(* CODESYS project XC300_NTPClient.project

Project tree, tasks and I/O mapping:
  XC303 : XC303, Eaton Automation, version 3.5.16.50
      unmapped channels: Output, Input
    application Application
      libraries: SysSocket23, * (System); SysCallback23, * (System); SysRtc23, * (System); Standard, 3.5.15.0 (System)
      task MainTask (cyclic, interval t#10ms, priority 1) calls PLC_PRG
      Global Variables/
        global variables Globale_Variablen
        global variables NetTime_Global
        global variables Variablen_Konfiguration
      POUs/
        Internal/
          function NetTime_Callback [ST]
          function NetTime_Concat_DT [ST]
          function NetTime_DayOfWeek [ST]
          function NetTime_SockClose [ST]
          function NetTime_SockCreate [ST]
          function block NetTime_Split_DT [IL]
        function block NetTime_RFC868_Client [ST]
        function block NetTime_RFC868_Server [ST]
        program PLC_PRG [ST]
  XV100 : XV100, Eaton Automation, version 3.5.16.60
    application Application
      libraries: SysSocket23, * (System); SysCallback23, * (System); SysRtc23, * (System); Standard, 3.5.15.0 (System)
      task MainTask (cyclic, interval t#10ms, priority 1) calls PLC_PRG
      Global Variables/
        global variables Globale_Variablen
        global variables NetTime_Global
        global variables Variablen_Konfiguration
      POUs/
        Internal/
          function NetTime_Callback [ST]
          function NetTime_Concat_DT [ST]
          function NetTime_DayOfWeek [ST]
          function NetTime_SockClose [ST]
          function NetTime_SockCreate [ST]
          function block NetTime_Split_DT [IL]
        function block NetTime_RFC868_Client [ST]
        function block NetTime_RFC868_Server [ST]
        program PLC_PRG [ST]
  XV300 : XV300, Eaton Automation, version 3.5.16.60
    application Application
      libraries: SysSocket23, * (System); SysCallback23, * (System); SysRtc23, * (System); Standard, 3.5.15.0 (System)
      task MainTask (cyclic, interval t#10ms, priority 1) calls PLC_PRG
      Global Variables/
        global variables Globale_Variablen
        global variables NetTime_Global
        global variables Variablen_Konfiguration
      POUs/
        Internal/
          function NetTime_Callback [ST]
          function NetTime_Concat_DT [ST]
          function NetTime_DayOfWeek [ST]
          function NetTime_SockClose [ST]
          function NetTime_SockCreate [ST]
          function block NetTime_Split_DT [IL]
        function block NetTime_RFC868_Client [ST]
        function block NetTime_RFC868_Server [ST]
        program PLC_PRG [ST]
*)

// XC303/Application/Global Variables/Globale_Variablen
VAR_GLOBAL
END_VAR

// XC303/Application/Global Variables/NetTime_Global
VAR_GLOBAL CONSTANT
	NetTime_striVersion 			: STRING := 'NTP V 1.0';							(* string with actual library version *)
	NetTime_iVersion_1_0		: INT;												(* variable to check compatibility *)
	NetTime_uiMaxSocketIndex 	: UINT := 10 ;										(* maximum count of sockets used in library *)
END_VAR
VAR_GLOBAL RETAIN
	NetTime_CallbackCounter : UINT ;
	NetTime_CallbackEVENT_STOPCounter : UINT ;
	NetTime_LastEvent : DWORD ;
	NetTime_LastFilter : DWORD ;
	NetTime_LastOwner : DWORD ;
END_VAR
VAR_GLOBAL
	NetTime_xCallbackRegistered : BOOL ;											(* callback function is registered *)
	NetTime_ar_udiSockets : ARRAY[1..NetTime_uiMaxSocketIndex] OF DINT ;	(* array with used socket IDs, 0 = empty *)
END_VAR

(*
Version		changes
1.0 			first version
*)

// XC303/Application/Global Variables/Variablen_Konfiguration
VAR_CONFIG
END_VAR

// XV100/Application/Global Variables/Globale_Variablen
VAR_GLOBAL
END_VAR

// XV100/Application/Global Variables/NetTime_Global
VAR_GLOBAL CONSTANT
	NetTime_striVersion 			: STRING := 'NTP V 1.0';							(* string with actual library version *)
	NetTime_iVersion_1_0		: INT;												(* variable to check compatibility *)
	NetTime_uiMaxSocketIndex 	: UINT := 10 ;										(* maximum count of sockets used in library *)
END_VAR
VAR_GLOBAL RETAIN
	NetTime_CallbackCounter : UINT ;
	NetTime_CallbackEVENT_STOPCounter : UINT ;
	NetTime_LastEvent : DWORD ;
	NetTime_LastFilter : DWORD ;
	NetTime_LastOwner : DWORD ;
END_VAR
VAR_GLOBAL
	NetTime_xCallbackRegistered : BOOL ;											(* callback function is registered *)
	NetTime_ar_udiSockets : ARRAY[1..NetTime_uiMaxSocketIndex] OF DINT ;	(* array with used socket IDs, 0 = empty *)
END_VAR

(*
Version		changes
1.0 			first version
*)

// XV100/Application/Global Variables/Variablen_Konfiguration
VAR_CONFIG
END_VAR

// XV300/Application/Global Variables/Globale_Variablen
VAR_GLOBAL
END_VAR

// XV300/Application/Global Variables/NetTime_Global
VAR_GLOBAL CONSTANT
	NetTime_striVersion 			: STRING := 'NTP V 1.0';							(* string with actual library version *)
	NetTime_iVersion_1_0		: INT;												(* variable to check compatibility *)
	NetTime_uiMaxSocketIndex 	: UINT := 10 ;										(* maximum count of sockets used in library *)
END_VAR
VAR_GLOBAL RETAIN
	NetTime_CallbackCounter : UINT ;
	NetTime_CallbackEVENT_STOPCounter : UINT ;
	NetTime_LastEvent : DWORD ;
	NetTime_LastFilter : DWORD ;
	NetTime_LastOwner : DWORD ;
END_VAR
VAR_GLOBAL
	NetTime_xCallbackRegistered : BOOL ;											(* callback function is registered *)
	NetTime_ar_udiSockets : ARRAY[1..NetTime_uiMaxSocketIndex] OF DINT ;	(* array with used socket IDs, 0 = empty *)
END_VAR

(*
Version		changes
1.0 			first version
*)

// XV300/Application/Global Variables/Variablen_Konfiguration
VAR_CONFIG
END_VAR

// XC303/Application/POUs/PLC_PRG
PROGRAM PLC_PRG
VAR
	FB_NetTime_RFC868_Client : NetTime_RFC868_Client ;
	FB_NetTime_RFC868_Server : NetTime_RFC868_Server ;
	FirstCall : BOOL := TRUE ;
END_VAR

(* Test of FB could be done with visualisation of XSoft *)

IF FirstCall THEN
	FB_NetTime_RFC868_Client.striIPAddress := '192.168.119.133' ;
	FB_NetTime_RFC868_Server.xEnable := 0 ;
END_IF
FirstCall := FALSE ;

FB_NetTime_RFC868_Client.xAskForTime;
FB_NetTime_RFC868_Client() ;

FB_NetTime_RFC868_Server() ;

END_PROGRAM

// XV100/Application/POUs/PLC_PRG
PROGRAM PLC_PRG
VAR
	FB_NetTime_RFC868_Client : NetTime_RFC868_Client ;
	FB_NetTime_RFC868_Server : NetTime_RFC868_Server ;
	FirstCall : BOOL := TRUE ;
END_VAR

(* Test of FB could be done with visualisation of XSoft *)

IF FirstCall THEN
	FB_NetTime_RFC868_Client.striIPAddress := '192.168.119.133' ;
	FB_NetTime_RFC868_Server.xEnable := TRUE ;
END_IF
FirstCall := FALSE ;

FB_NetTime_RFC868_Client.xAskForTime;
FB_NetTime_RFC868_Client() ;

FB_NetTime_RFC868_Server() ;

END_PROGRAM

// XV300/Application/POUs/PLC_PRG
PROGRAM PLC_PRG
VAR
	FB_NetTime_RFC868_Client : NetTime_RFC868_Client ;
	FB_NetTime_RFC868_Server : NetTime_RFC868_Server ;
	FirstCall : BOOL := TRUE ;
END_VAR

(* Test of FB could be done with visualisation of XSoft *)

IF FirstCall THEN
	FB_NetTime_RFC868_Client.striIPAddress := '192.168.119.248' ;
	FB_NetTime_RFC868_Server.xEnable := TRUE ;
END_IF
FirstCall := FALSE ;

FB_NetTime_RFC868_Client.xAskForTime;
FB_NetTime_RFC868_Client() ;

FB_NetTime_RFC868_Server() ;

END_PROGRAM

// XC303/Application/POUs/NetTime_RFC868_Client
FUNCTION_BLOCK NetTime_RFC868_Client
(* this FB is a client for time request to a server using a protocol described in RFC868 / UDP *)

VAR_INPUT
	striIPAddress : STRING(15) ; 				(* IP-address of th time server i.e '192.168.0.1' *)
	uiLocalPort : UINT := 1025 ;				(* local ethernet port 1-65535 see RFC1700 for assigned ports *)
	xAskForTime : BOOL ;						(* rising edge send a time request to the server *)
	siGMTOffset : SINT := 1 ;					(* time offset in h for local time-zone (-12..+12) i.e. +1 for Berlin *)
	xSummerWinterTime : BOOL := TRUE ;	(* consider Summertime from last sunday of march at 02:00 a.m.GMT to last sunday of october at 02:00 a.m.GMT *)
	xSetRTC : BOOL ;							(* set the local Real-Time-Clock to the received time from server *)
END_VAR

VAR_OUTPUT
	dtReceivedDateTime : DT := DATE_AND_TIME#2000-01-01-00:00:00 ;		(* received Date and Time from server *)
	uiReceivedSecond : UINT ;				(* received second from server (0..59) *)
	uiReceivedMinute : UINT ;				(* received minute from server (0..59) *)
	uiReceivedHour : UINT ;					(* received hour from server (0..23) *)
	uiReceivedDay : UINT :=1 ;				(* received Day from server (1..31) *)
	uiReceivedMonth : UINT :=1 ;				(* received Month from server (1..12) *)
	uiReceivedYear : UINT :=2000 ;			(* received year from server (2000..2092) *)
	uiReceivedDayOfWeek : UINT := 6 ;		(* received weekday. (1=Monday .. 7=Sunday) *)
	xSummerTime : BOOL ;					(* received Time is Summertime *)
	xActive : BOOL ;							(* waiting for an answer of the time server *)
	xError : BOOL ;							(* last request generate an error - look "uiErrornumber" for reason *)
	uiErrorNumber : UINT ;					(* reason for the last error
		0 = No error
		1 = Ethernet socket could not opend 
		2 = Ethernet socket could not binded
		3 = Transmit time request error
		4 = Ethernet receive error
		5 = Timeout - no answer from timeserver in the space of 5s *)
END_VAR

VAR
	xAskForTimeOld : BOOL ;
	iSocketIndex : UINT ;
	xBindSocket : BOOL ;
	diTraNr : DINT ;
	udiTime : UDINT ;
	struSOCKADDRESS_Receive : SOCKADDRESS ;
	diRecNr : DINT ;
	diIO : DINT ;
	dwParameterIO : DWORD ;
	arReceiveData : ARRAY[0..3] OF BYTE ;
	xRecIP : BOOL ;
	struInADDR_TimeServer : INADDR;
	striTimeServerIPAddress : STRING;

	TON_Timeout : TON := (PT:=T#5s) ;

	uiRemotePort : UINT := 37 ;
	struSOCKADDRESS_Bind : SOCKADDRESS ;
	struSOCKADDRESS_Transmit : SOCKADDRESS ;
	dwReceiveData : DWORD ;
	udiGMTSecondsSince1970 : UDINT ;
	i : USINT ;

	Split_DT : NetTime_Split_DT ;

	uiDayStartSummertime : UINT ;
	uiDayEndSummertime : UINT ;

	dtStartSummertime : DT ;
	dtEndSummertime : DT ;

	struSOCKADDRESS_Connect : SOCKADDRESS ;
	xSysSockConnect : BOOL ;
END_VAR

IF xActive THEN
	IF NetTime_ar_udiSockets[iSocketIndex] > 0 THEN
		(* waiting for an answer of the time-server *)
		(* is any data received *)
		diIO := SysSockIoctl(NetTime_ar_udiSockets[iSocketIndex], SOCKET_FIONREAD, ADR(dwParameterIO)); (* get num chars available to read *)
		IF dwParameterIO <> 0 THEN
			diRecNr := SysSockRecvFrom(NetTime_ar_udiSockets[iSocketIndex], ADR(arReceiveData), SIZEOF(arReceiveData), 0,
											 ADR(struSOCKADDRESS_Receive), SIZEOF(struSOCKADDRESS_Receive));
			IF diRecNr = -1 THEN
				uiErrorNumber := 4 ;
			ELSE
				(* check receive IP Address *)
				struInADDR_TimeServer.s_addr := struSOCKADDRESS_Receive.sin_addr ;
				xRecIP:=SysSockInetNtoa(struInADDR_TimeServer, striTimeServerIPAddress, SIZEOF(striTimeServerIPAddress)) ;
				IF struSOCKADDRESS_Receive.sin_addr = struSOCKADDRESS_Transmit.sin_addr THEN
					(* answer is coming from requested timeserver *)
					(* interpret received data *)
					(* change byte orientation *)
					dwReceiveData := 0 ;
					FOR i := 0 TO 3 DO
						dwReceiveData := SHL(dwReceiveData,8) ;
						dwReceiveData := dwReceiveData OR BYTE_TO_DWORD(arReceiveData[i]) ;
					END_FOR
					(* dwReceiveData = seconds after 1.1.1900 00:00:00 *)
					IF DWORD_TO_UDINT(dwReceiveData) >= UDINT#2208988800 THEN
						udiGMTSecondsSince1970 := DWORD_TO_UDINT(dwReceiveData) - UDINT#2208988800 ;
					ELSE
						udiGMTSecondsSince1970 := DWORD_TO_UDINT(dwReceiveData) + UDINT#2208988800 ;
					END_IF
					dtReceivedDateTime := UDINT_TO_DT(udiGMTSecondsSince1970+(UINT#3600*SINT_TO_DINT(siGMTOffset))) ;
	
					Split_DT(
						InputDT:=dtReceivedDateTime ,
						uiSecond=>uiReceivedSecond ,
						uiMinute=>uiReceivedMinute ,
						uiHour=>uiReceivedHour ,
						uiDay=>uiReceivedDay ,
						uiMonth=>uiReceivedMonth ,
						uiYear=>uiReceivedYear );
	
					uiReceivedDayOfWeek := NetTime_DayOfWeek(uiReceivedDay,uiReceivedMonth,uiReceivedYear) ;
	
					IF xSummerWinterTime THEN
						(* check if the received time is in summertime interval
						last sunday of march at 2:00 a.m. to last sunday of october at 2:00 a.m. *)
						uiDayStartSummertime := 31-NetTime_DayOfWeek(31,3,uiReceivedYear) ;
						uiDayEndSummertime := 31-NetTime_DayOfWeek(31,10,uiReceivedYear) ;
						dtStartSummertime := NetTime_Concat_DT(0,0,2,uiDayStartSummertime,3,uiReceivedYear) ;
						dtEndSummertime := NetTime_Concat_DT(0,0,2,uiDayEndSummertime,10,uiReceivedYear) ;
						xSummerTime := (dtReceivedDateTime>dtStartSummertime) AND (dtReceivedDateTime<dtEndSummertime) ;
						IF xSummerTime THEN
							(* add 1 hour to GMT time *)
							dtReceivedDateTime := UDINT_TO_DT(DT_TO_UDINT(dtReceivedDateTime) + UDINT#3600) ;
							Split_DT(
								InputDT:=dtReceivedDateTime ,
								uiSecond=>uiReceivedSecond ,
								uiMinute=>uiReceivedMinute ,
								uiHour=>uiReceivedHour ,
								uiDay=>uiReceivedDay ,
								uiMonth=>uiReceivedMonth ,
								uiYear=>uiReceivedYear );
						END_IF
					END_IF
	
					IF xSetRTC THEN
						(* set the local RTC to the received time *)
						SysRtcSetTime(dtReceivedDateTime) ;
					END_IF
	
					(* close socket *)
					NetTime_SockClose(iSocketIndex) ;
					xActive := FALSE ;
				END_IF
			END_IF
	
		ELSE
			TON_Timeout();
			IF TON_Timeout.Q THEN
				uiErrorNumber := 5 ;
				NetTime_SockClose(iSocketIndex) ;
				xActive := FALSE ;
				TON_Timeout(IN:=FALSE) ;
			END_IF
		END_IF
	ELSE
		(* Socketindex is no longer valid! Perhaps PLC has stopt and socket has closed *)
		uiErrorNumber := 5 ;
		xActive := FALSE ;
	END_IF
ELSE
	(* waiting for a new request *)
	IF xAskForTime AND NOT xAskForTimeOld THEN
		(* start time request *)
		dtReceivedDateTime := DATE_AND_TIME#2000-01-01-00:00:00 ;
		uiReceivedSecond := 0 ;
		uiReceivedMinute := 0 ;
		uiReceivedHour := 0 ;
		uiReceivedDay := 1 ;
		uiReceivedMonth := 1 ;
		uiReceivedYear := 2000 ;
		uiReceivedDayOfWeek := 6 ;
		xError := FALSE ;
		uiErrorNumber := 0;
	
		(* create a new  datagram-socket *)
		iSocketIndex := NetTime_SockCreate(SOCKET_AF_INET,SOCKET_DGRAM,0);
		IF iSocketIndex > 0 THEN
			(* Bind the socket to the local port *)
			struSOCKADDRESS_Bind.sin_family := SOCKET_AF_INET; (* internetwork: UDP, TCP, etc. *)
			struSOCKADDRESS_Bind.sin_addr := SysSockHtonl(SOCKET_INADDR_ANY) ;
			struSOCKADDRESS_Bind.sin_port := SysSockHtons(uiLocalPort);
			xBindSocket := SysSockBind(NetTime_ar_udiSockets[iSocketIndex], ADR(struSOCKADDRESS_Bind), SIZEOF(struSOCKADDRESS_Bind));
			IF  xBindSocket THEN
				(* UDP: send a time request to the time server *)
				struSOCKADDRESS_Transmit.sin_family := SOCKET_AF_INET; (* internetwork: UDP, TCP, etc. *)
				struSOCKADDRESS_Transmit.sin_addr := SysSockInetAddr(striIPAddress);
				struSOCKADDRESS_Transmit.sin_port := SysSockHtons(uiRemotePort);
				diTraNr := SysSockSendTo(NetTime_ar_udiSockets[iSocketIndex] , ADR(udiTime), 4,0,
							ADR(struSOCKADDRESS_Transmit), SIZEOF(struSOCKADDRESS_Transmit));
				IF diTraNr < 0 THEN
					uiErrorNumber := 3 ;
					NetTime_SockClose(iSocketIndex) ;
				ELSE
					(* start timeout timer *)
					TON_Timeout(IN:=FALSE) ;
					TON_Timeout(IN:=TRUE) ;
					xActive := TRUE ;
				END_IF
			ELSE
				NetTime_SockClose(iSocketIndex);
				uiErrorNumber := 2 ;
			END_IF
		ELSE
			uiErrorNumber := 1 ;
			NetTime_SockClose(iSocketIndex);
		END_IF
	END_IF
END_IF

xAskForTimeOld := xAskForTime ;
xError := uiErrorNumber<>0 ;

END_FUNCTION_BLOCK

// XC303/Application/POUs/Internal/NetTime_DayOfWeek
FUNCTION NetTime_DayOfWeek : UINT
(* function calculate the day of week from input date (1=Monday .. 7=Sunday) *)
VAR_INPUT
	uiDay : UINT ;		(* day of date (1..31) *)
	uiMonth : UINT ;	(* month of date (1..12) *)
	uiYear :UINT ;		(* year of date (2000..2092) *)
END_VAR

VAR
	uiLastDigitOfYear : UINT ;
	uiQuarterOfLastDigitOfYear : UINT ;
	uiMonthCode : UINT ;
	xLeapyear : BOOL ;
END_VAR

uiLastDigitOfYear := uiYear MOD 100 ;
xLeapyear := (uiYear MOD 4 = 0) ;
uiQuarterOfLastDigitOfYear := uiLastDigitOfYear / 4 ;
CASE uiMonth OF
	1:	uiMonthCode := 6 ;
	2:	uiMonthCode := 2 ;
	3:	uiMonthCode := 2 ;
	4:	uiMonthCode := 5 ;
	5:	uiMonthCode := 0 ;
	6:	uiMonthCode := 3 ;
	7:	uiMonthCode := 5 ;
	8:	uiMonthCode := 1 ;
	9:	uiMonthCode := 4 ;
	10:	uiMonthCode := 6 ;
	11:	uiMonthCode := 2 ;
	12:	uiMonthCode := 4 ;
END_CASE
NetTime_DayOfWeek := (uiLastDigitOfYear + uiQuarterOfLastDigitOfYear + uiMonthCode + uiDay) MOD 7 ;
IF xLeapyear AND (uiMonth<3) THEN
	NetTime_DayOfWeek := NetTime_DayOfWeek - 1 ;
END_IF

END_FUNCTION

// XV100/Application/POUs/Internal/NetTime_DayOfWeek
FUNCTION NetTime_DayOfWeek : UINT
(* function calculate the day of week from input date (1=Monday .. 7=Sunday) *)
VAR_INPUT
	uiDay : UINT ;		(* day of date (1..31) *)
	uiMonth : UINT ;	(* month of date (1..12) *)
	uiYear :UINT ;		(* year of date (2000..2092) *)
END_VAR

VAR
	uiLastDigitOfYear : UINT ;
	uiQuarterOfLastDigitOfYear : UINT ;
	uiMonthCode : UINT ;
	xLeapyear : BOOL ;
END_VAR

uiLastDigitOfYear := uiYear MOD 100 ;
xLeapyear := (uiYear MOD 4 = 0) ;
uiQuarterOfLastDigitOfYear := uiLastDigitOfYear / 4 ;
CASE uiMonth OF
	1:	uiMonthCode := 6 ;
	2:	uiMonthCode := 2 ;
	3:	uiMonthCode := 2 ;
	4:	uiMonthCode := 5 ;
	5:	uiMonthCode := 0 ;
	6:	uiMonthCode := 3 ;
	7:	uiMonthCode := 5 ;
	8:	uiMonthCode := 1 ;
	9:	uiMonthCode := 4 ;
	10:	uiMonthCode := 6 ;
	11:	uiMonthCode := 2 ;
	12:	uiMonthCode := 4 ;
END_CASE
NetTime_DayOfWeek := (uiLastDigitOfYear + uiQuarterOfLastDigitOfYear + uiMonthCode + uiDay) MOD 7 ;
IF xLeapyear AND (uiMonth<3) THEN
	NetTime_DayOfWeek := NetTime_DayOfWeek - 1 ;
END_IF

END_FUNCTION

// XV300/Application/POUs/Internal/NetTime_DayOfWeek
FUNCTION NetTime_DayOfWeek : UINT
(* function calculate the day of week from input date (1=Monday .. 7=Sunday) *)
VAR_INPUT
	uiDay : UINT ;		(* day of date (1..31) *)
	uiMonth : UINT ;	(* month of date (1..12) *)
	uiYear :UINT ;		(* year of date (2000..2092) *)
END_VAR

VAR
	uiLastDigitOfYear : UINT ;
	uiQuarterOfLastDigitOfYear : UINT ;
	uiMonthCode : UINT ;
	xLeapyear : BOOL ;
END_VAR

uiLastDigitOfYear := uiYear MOD 100 ;
xLeapyear := (uiYear MOD 4 = 0) ;
uiQuarterOfLastDigitOfYear := uiLastDigitOfYear / 4 ;
CASE uiMonth OF
	1:	uiMonthCode := 6 ;
	2:	uiMonthCode := 2 ;
	3:	uiMonthCode := 2 ;
	4:	uiMonthCode := 5 ;
	5:	uiMonthCode := 0 ;
	6:	uiMonthCode := 3 ;
	7:	uiMonthCode := 5 ;
	8:	uiMonthCode := 1 ;
	9:	uiMonthCode := 4 ;
	10:	uiMonthCode := 6 ;
	11:	uiMonthCode := 2 ;
	12:	uiMonthCode := 4 ;
END_CASE
NetTime_DayOfWeek := (uiLastDigitOfYear + uiQuarterOfLastDigitOfYear + uiMonthCode + uiDay) MOD 7 ;
IF xLeapyear AND (uiMonth<3) THEN
	NetTime_DayOfWeek := NetTime_DayOfWeek - 1 ;
END_IF

END_FUNCTION

// XC303/Application/POUs/Internal/NetTime_Concat_DT
FUNCTION NetTime_Concat_DT : DT
(* FB concat input values to the DT data type. There is no check for validity of the input data!
The input data must between 01.01.2000 00:00:00  and 31.12.2092 23:59:59 *)
VAR_INPUT
	uiSecond : UINT ;	(* second of DT (0..59) *)
	uiMinute : UINT ;	(* minute of DT (0..59) *)
	uiHour : UINT ;	(* hour of DT (1..23) *)
	uiDay : UINT ;		(* day of DT (1..31) *)
	uiMonth : UINT ;	(* month of DT (1..12) *)
	uiYear :UINT ;		(* year of DT (2000..2092) *)
END_VAR

VAR
	xLeapYear : BOOL ;
	uiYearsSince1970 : UINT ;
	uiCountOfLeapDays : UINT ;
	uiDaysInActualYear : UINT ;
	udiSecondsSince1970 : UDINT ;
END_VAR

CASE uiMonth OF
	1:	uiDaysInActualYear := 0 ;
	2:	uiDaysInActualYear := 31;
	3:	uiDaysInActualYear := 59 ;
	4:	uiDaysInActualYear := 90 ;
	5:	uiDaysInActualYear := 120 ;
	6:	uiDaysInActualYear := 151 ;
	7:	uiDaysInActualYear := 181 ;
	8:	uiDaysInActualYear := 212 ;
	9:	uiDaysInActualYear := 243 ;
	10:	uiDaysInActualYear := 273 ;
	11:	uiDaysInActualYear := 304 ;
	12:	uiDaysInActualYear := 334 ;
END_CASE
uiDaysInActualYear := uiDaysInActualYear + uiday ;

uiYearsSince1970 := uiYear - 1970 ;
xLeapYear := (uiYear MOD 4) = 0 ;
uiCountOfLeapDays := (uiYearsSince1970 - 2) / 4 ;
IF (xLeapYear) AND (uiMonth<3) THEN
	uiCountOfLeapDays := uiCountOfLeapDays - 1 ;
END_IF

udiSecondsSince1970 :=
		(UINT_TO_UDINT(uiYearsSince1970) * UDINT#31536000)
	+ 	(UINT_TO_UDINT(uiDaysInActualYear+uiCountOfLeapDays) * UDINT#86400)
	+	(UINT_TO_UDINT(uiHour) * UDINT#3600)
	+	(UINT_TO_UDINT(uiMinute) * UDINT#60)
	+	(UINT_TO_UDINT(uiSecond)) ;

NetTime_Concat_DT := UDINT_TO_DT(udiSecondsSince1970) ;

END_FUNCTION

// XV100/Application/POUs/Internal/NetTime_Concat_DT
FUNCTION NetTime_Concat_DT : DT
(* FB concat input values to the DT data type. There is no check for validity of the input data!
The input data must between 01.01.2000 00:00:00  and 31.12.2092 23:59:59 *)
VAR_INPUT
	uiSecond : UINT ;	(* second of DT (0..59) *)
	uiMinute : UINT ;	(* minute of DT (0..59) *)
	uiHour : UINT ;	(* hour of DT (1..23) *)
	uiDay : UINT ;		(* day of DT (1..31) *)
	uiMonth : UINT ;	(* month of DT (1..12) *)
	uiYear :UINT ;		(* year of DT (2000..2092) *)
END_VAR

VAR
	xLeapYear : BOOL ;
	uiYearsSince1970 : UINT ;
	uiCountOfLeapDays : UINT ;
	uiDaysInActualYear : UINT ;
	udiSecondsSince1970 : UDINT ;
END_VAR

CASE uiMonth OF
	1:	uiDaysInActualYear := 0 ;
	2:	uiDaysInActualYear := 31;
	3:	uiDaysInActualYear := 59 ;
	4:	uiDaysInActualYear := 90 ;
	5:	uiDaysInActualYear := 120 ;
	6:	uiDaysInActualYear := 151 ;
	7:	uiDaysInActualYear := 181 ;
	8:	uiDaysInActualYear := 212 ;
	9:	uiDaysInActualYear := 243 ;
	10:	uiDaysInActualYear := 273 ;
	11:	uiDaysInActualYear := 304 ;
	12:	uiDaysInActualYear := 334 ;
END_CASE
uiDaysInActualYear := uiDaysInActualYear + uiday ;

uiYearsSince1970 := uiYear - 1970 ;
xLeapYear := (uiYear MOD 4) = 0 ;
uiCountOfLeapDays := (uiYearsSince1970 - 2) / 4 ;
IF (xLeapYear) AND (uiMonth<3) THEN
	uiCountOfLeapDays := uiCountOfLeapDays - 1 ;
END_IF

udiSecondsSince1970 :=
		(UINT_TO_UDINT(uiYearsSince1970) * UDINT#31536000)
	+ 	(UINT_TO_UDINT(uiDaysInActualYear+uiCountOfLeapDays) * UDINT#86400)
	+	(UINT_TO_UDINT(uiHour) * UDINT#3600)
	+	(UINT_TO_UDINT(uiMinute) * UDINT#60)
	+	(UINT_TO_UDINT(uiSecond)) ;

NetTime_Concat_DT := UDINT_TO_DT(udiSecondsSince1970) ;

END_FUNCTION

// XV300/Application/POUs/Internal/NetTime_Concat_DT
FUNCTION NetTime_Concat_DT : DT
(* FB concat input values to the DT data type. There is no check for validity of the input data!
The input data must between 01.01.2000 00:00:00  and 31.12.2092 23:59:59 *)
VAR_INPUT
	uiSecond : UINT ;	(* second of DT (0..59) *)
	uiMinute : UINT ;	(* minute of DT (0..59) *)
	uiHour : UINT ;	(* hour of DT (1..23) *)
	uiDay : UINT ;		(* day of DT (1..31) *)
	uiMonth : UINT ;	(* month of DT (1..12) *)
	uiYear :UINT ;		(* year of DT (2000..2092) *)
END_VAR

VAR
	xLeapYear : BOOL ;
	uiYearsSince1970 : UINT ;
	uiCountOfLeapDays : UINT ;
	uiDaysInActualYear : UINT ;
	udiSecondsSince1970 : UDINT ;
END_VAR

CASE uiMonth OF
	1:	uiDaysInActualYear := 0 ;
	2:	uiDaysInActualYear := 31;
	3:	uiDaysInActualYear := 59 ;
	4:	uiDaysInActualYear := 90 ;
	5:	uiDaysInActualYear := 120 ;
	6:	uiDaysInActualYear := 151 ;
	7:	uiDaysInActualYear := 181 ;
	8:	uiDaysInActualYear := 212 ;
	9:	uiDaysInActualYear := 243 ;
	10:	uiDaysInActualYear := 273 ;
	11:	uiDaysInActualYear := 304 ;
	12:	uiDaysInActualYear := 334 ;
END_CASE
uiDaysInActualYear := uiDaysInActualYear + uiday ;

uiYearsSince1970 := uiYear - 1970 ;
xLeapYear := (uiYear MOD 4) = 0 ;
uiCountOfLeapDays := (uiYearsSince1970 - 2) / 4 ;
IF (xLeapYear) AND (uiMonth<3) THEN
	uiCountOfLeapDays := uiCountOfLeapDays - 1 ;
END_IF

udiSecondsSince1970 :=
		(UINT_TO_UDINT(uiYearsSince1970) * UDINT#31536000)
	+ 	(UINT_TO_UDINT(uiDaysInActualYear+uiCountOfLeapDays) * UDINT#86400)
	+	(UINT_TO_UDINT(uiHour) * UDINT#3600)
	+	(UINT_TO_UDINT(uiMinute) * UDINT#60)
	+	(UINT_TO_UDINT(uiSecond)) ;

NetTime_Concat_DT := UDINT_TO_DT(udiSecondsSince1970) ;

END_FUNCTION

// XC303/Application/POUs/Internal/NetTime_SockClose
FUNCTION NetTime_SockClose : BOOL
(* close the socket and delete it out of the global array.TRUE if function is successful *)
VAR_INPUT
	iSocketIndex : UINT ;	(* Index of tthe socket id in the global field to close. Get from function "NetTime_SockCreate" *)
END_VAR

IF iSocketIndex>0 AND iSocketIndex<=NetTime_uiMaxSocketIndex THEN
	NetTime_SockClose := SysSockClose(NetTime_ar_udiSockets[iSocketIndex]) ;
	IF NetTime_SockClose THEN
		NetTime_ar_udiSockets[iSocketIndex] := 0 ;
	END_IF
END_IF

END_FUNCTION

// XV100/Application/POUs/Internal/NetTime_SockClose
FUNCTION NetTime_SockClose : BOOL
(* close the socket and delete it out of the global array.TRUE if function is successful *)
VAR_INPUT
	iSocketIndex : UINT ;	(* Index of tthe socket id in the global field to close. Get from function "NetTime_SockCreate" *)
END_VAR

IF iSocketIndex>0 AND iSocketIndex<=NetTime_uiMaxSocketIndex THEN
	NetTime_SockClose := SysSockClose(NetTime_ar_udiSockets[iSocketIndex]) ;
	IF NetTime_SockClose THEN
		NetTime_ar_udiSockets[iSocketIndex] := 0 ;
	END_IF
END_IF

END_FUNCTION

// XV300/Application/POUs/Internal/NetTime_SockClose
FUNCTION NetTime_SockClose : BOOL
(* close the socket and delete it out of the global array.TRUE if function is successful *)
VAR_INPUT
	iSocketIndex : UINT ;	(* Index of tthe socket id in the global field to close. Get from function "NetTime_SockCreate" *)
END_VAR

IF iSocketIndex>0 AND iSocketIndex<=NetTime_uiMaxSocketIndex THEN
	NetTime_SockClose := SysSockClose(NetTime_ar_udiSockets[iSocketIndex]) ;
	IF NetTime_SockClose THEN
		NetTime_ar_udiSockets[iSocketIndex] := 0 ;
	END_IF
END_IF

END_FUNCTION

// XC303/Application/POUs/Internal/NetTime_SockCreate
FUNCTION NetTime_SockCreate : INT
(* create e new socket and save ID in global array. function supply the id of the socket  *)
VAR_INPUT
	diAddressFamily : DINT ;	(* family of the addres. i.e. SOCKET_AF_INET for TCP/UDP *)
	diType : DINT ;				(* type of the address. i.e. SOCKET_DGRAM *)
	diProtocol : DINT ;			(* protocol of the address i.e. SOCKET_IPPROTO_IP *)
END_VAR
VAR
	uiIndex : UINT ;
	SockCreate : DINT ;
END_VAR

(* register callback function to close all sockets on PLC event STOP *)
IF NOT NetTime_xCallbackRegistered THEN
	SysCallbackRegister(ADR(NetTime_Callback),EVENT_STOP) ;
	NetTime_xCallbackRegistered := TRUE ;
END_IF

(* look for an empty field in the global socket array *)
uiIndex := 1 ;
WHILE NetTime_ar_udiSockets[uiIndex] <> 0 DO
	uiIndex := uiIndex + 1 ;
	IF  uiIndex > NetTime_uiMaxSocketIndex THEN
		EXIT ;
	END_IF
END_WHILE

IF uiIndex > NetTime_uiMaxSocketIndex THEN
	(* it is not possible to create a new socket *)
	NetTime_SockCreate := -1 ;
ELSE
	(* try to create a new socket *)
	SockCreate := SysSockCreate(diAddressFamily,diType,diProtocol) ;
	IF SockCreate <> SOCKET_INVALID THEN
		(* save the socket ID in the global array *)
		NetTime_ar_udiSockets[uiIndex] := SockCreate ;
		NetTime_SockCreate := uiIndex ;
	END_IF
END_IF

END_FUNCTION

// XC303/Application/POUs/Internal/NetTime_Callback
FUNCTION NetTime_Callback : DWORD
(* this function is called from RTS on event STOP to close all sockets *)
VAR_INPUT
	dwEvent : DWORD ;
	dwFilter : DWORD ;
	dwOwner : DWORD ;
END_VAR

VAR
	uiIndex : UINT ;
END_VAR

(* Close all sockets on STOP *)
NetTime_LastEvent := dwEvent ;
NetTime_LastFilter := dwFilter ;
NetTime_LastOwner := dwOwner ;
NetTime_CallbackCounter := NetTime_CallbackCounter + 1;
IF dwEvent = EVENT_STOP THEN
	NetTime_CallbackEVENT_STOPCounter := NetTime_CallbackEVENT_STOPCounter + 1;
END_IF
FOR uiIndex := 1 TO NetTime_uiMaxSocketIndex DO
	IF NetTime_ar_udiSockets[uiIndex] <> 0 THEN
		SysSockClose(NetTime_ar_udiSockets[uiIndex]) ;
		NetTime_ar_udiSockets[uiIndex] := 0 ;
	END_IF
END_FOR

END_FUNCTION

// XV100/Application/POUs/Internal/NetTime_Callback
FUNCTION NetTime_Callback : DWORD
(* this function is called from RTS on event STOP to close all sockets *)
VAR_INPUT
	dwEvent : DWORD ;
	dwFilter : DWORD ;
	dwOwner : DWORD ;
END_VAR

VAR
	uiIndex : UINT ;
END_VAR

(* Close all sockets on STOP *)
NetTime_LastEvent := dwEvent ;
NetTime_LastFilter := dwFilter ;
NetTime_LastOwner := dwOwner ;
NetTime_CallbackCounter := NetTime_CallbackCounter + 1;
IF dwEvent = EVENT_STOP THEN
	NetTime_CallbackEVENT_STOPCounter := NetTime_CallbackEVENT_STOPCounter + 1;
END_IF
FOR uiIndex := 1 TO NetTime_uiMaxSocketIndex DO
	IF NetTime_ar_udiSockets[uiIndex] <> 0 THEN
		SysSockClose(NetTime_ar_udiSockets[uiIndex]) ;
		NetTime_ar_udiSockets[uiIndex] := 0 ;
	END_IF
END_FOR

END_FUNCTION

// XV300/Application/POUs/Internal/NetTime_Callback
FUNCTION NetTime_Callback : DWORD
(* this function is called from RTS on event STOP to close all sockets *)
VAR_INPUT
	dwEvent : DWORD ;
	dwFilter : DWORD ;
	dwOwner : DWORD ;
END_VAR

VAR
	uiIndex : UINT ;
END_VAR

(* Close all sockets on STOP *)
NetTime_LastEvent := dwEvent ;
NetTime_LastFilter := dwFilter ;
NetTime_LastOwner := dwOwner ;
NetTime_CallbackCounter := NetTime_CallbackCounter + 1;
IF dwEvent = EVENT_STOP THEN
	NetTime_CallbackEVENT_STOPCounter := NetTime_CallbackEVENT_STOPCounter + 1;
END_IF
FOR uiIndex := 1 TO NetTime_uiMaxSocketIndex DO
	IF NetTime_ar_udiSockets[uiIndex] <> 0 THEN
		SysSockClose(NetTime_ar_udiSockets[uiIndex]) ;
		NetTime_ar_udiSockets[uiIndex] := 0 ;
	END_IF
END_FOR

END_FUNCTION

// XV100/Application/POUs/Internal/NetTime_SockCreate
FUNCTION NetTime_SockCreate : INT
(* create e new socket and save ID in global array. function supply the id of the socket  *)
VAR_INPUT
	diAddressFamily : DINT ;	(* family of the addres. i.e. SOCKET_AF_INET for TCP/UDP *)
	diType : DINT ;				(* type of the address. i.e. SOCKET_DGRAM *)
	diProtocol : DINT ;			(* protocol of the address i.e. SOCKET_IPPROTO_IP *)
END_VAR
VAR
	uiIndex : UINT ;
	SockCreate : DINT ;
END_VAR

(* register callback function to close all sockets on PLC event STOP *)
IF NOT NetTime_xCallbackRegistered THEN
	SysCallbackRegister(ADR(NetTime_Callback),EVENT_STOP) ;
	NetTime_xCallbackRegistered := TRUE ;
END_IF

(* look for an empty field in the global socket array *)
uiIndex := 1 ;
WHILE NetTime_ar_udiSockets[uiIndex] <> 0 DO
	uiIndex := uiIndex + 1 ;
	IF  uiIndex > NetTime_uiMaxSocketIndex THEN
		EXIT ;
	END_IF
END_WHILE

IF uiIndex > NetTime_uiMaxSocketIndex THEN
	(* it is not possible to create a new socket *)
	NetTime_SockCreate := -1 ;
ELSE
	(* try to create a new socket *)
	SockCreate := SysSockCreate(diAddressFamily,diType,diProtocol) ;
	IF SockCreate <> SOCKET_INVALID THEN
		(* save the socket ID in the global array *)
		NetTime_ar_udiSockets[uiIndex] := SockCreate ;
		NetTime_SockCreate := uiIndex ;
	END_IF
END_IF

END_FUNCTION

// XV300/Application/POUs/Internal/NetTime_SockCreate
FUNCTION NetTime_SockCreate : INT
(* create e new socket and save ID in global array. function supply the id of the socket  *)
VAR_INPUT
	diAddressFamily : DINT ;	(* family of the addres. i.e. SOCKET_AF_INET for TCP/UDP *)
	diType : DINT ;				(* type of the address. i.e. SOCKET_DGRAM *)
	diProtocol : DINT ;			(* protocol of the address i.e. SOCKET_IPPROTO_IP *)
END_VAR
VAR
	uiIndex : UINT ;
	SockCreate : DINT ;
END_VAR

(* register callback function to close all sockets on PLC event STOP *)
IF NOT NetTime_xCallbackRegistered THEN
	SysCallbackRegister(ADR(NetTime_Callback),EVENT_STOP) ;
	NetTime_xCallbackRegistered := TRUE ;
END_IF

(* look for an empty field in the global socket array *)
uiIndex := 1 ;
WHILE NetTime_ar_udiSockets[uiIndex] <> 0 DO
	uiIndex := uiIndex + 1 ;
	IF  uiIndex > NetTime_uiMaxSocketIndex THEN
		EXIT ;
	END_IF
END_WHILE

IF uiIndex > NetTime_uiMaxSocketIndex THEN
	(* it is not possible to create a new socket *)
	NetTime_SockCreate := -1 ;
ELSE
	(* try to create a new socket *)
	SockCreate := SysSockCreate(diAddressFamily,diType,diProtocol) ;
	IF SockCreate <> SOCKET_INVALID THEN
		(* save the socket ID in the global array *)
		NetTime_ar_udiSockets[uiIndex] := SockCreate ;
		NetTime_SockCreate := uiIndex ;
	END_IF
END_IF

END_FUNCTION

// XV100/Application/POUs/NetTime_RFC868_Client
FUNCTION_BLOCK NetTime_RFC868_Client
(* this FB is a client for time request to a server using a protocol described in RFC868 / UDP *)

VAR_INPUT
	striIPAddress : STRING(15) ; 				(* IP-address of th time server i.e '192.168.0.1' *)
	uiLocalPort : UINT := 1025 ;				(* local ethernet port 1-65535 see RFC1700 for assigned ports *)
	xAskForTime : BOOL ;						(* rising edge send a time request to the server *)
	siGMTOffset : SINT := 1 ;					(* time offset in h for local time-zone (-12..+12) i.e. +1 for Berlin *)
	xSummerWinterTime : BOOL := TRUE ;	(* consider Summertime from last sunday of march at 02:00 a.m.GMT to last sunday of october at 02:00 a.m.GMT *)
	xSetRTC : BOOL ;							(* set the local Real-Time-Clock to the received time from server *)
END_VAR

VAR_OUTPUT
	dtReceivedDateTime : DT := DATE_AND_TIME#2000-01-01-00:00:00 ;		(* received Date and Time from server *)
	uiReceivedSecond : UINT ;				(* received second from server (0..59) *)
	uiReceivedMinute : UINT ;				(* received minute from server (0..59) *)
	uiReceivedHour : UINT ;					(* received hour from server (0..23) *)
	uiReceivedDay : UINT :=1 ;				(* received Day from server (1..31) *)
	uiReceivedMonth : UINT :=1 ;				(* received Month from server (1..12) *)
	uiReceivedYear : UINT :=2000 ;			(* received year from server (2000..2092) *)
	uiReceivedDayOfWeek : UINT := 6 ;		(* received weekday. (1=Monday .. 7=Sunday) *)
	xSummerTime : BOOL ;					(* received Time is Summertime *)
	xActive : BOOL ;							(* waiting for an answer of the time server *)
	xError : BOOL ;							(* last request generate an error - look "uiErrornumber" for reason *)
	uiErrorNumber : UINT ;					(* reason for the last error
		0 = No error
		1 = Ethernet socket could not opend 
		2 = Ethernet socket could not binded
		3 = Transmit time request error
		4 = Ethernet receive error
		5 = Timeout - no answer from timeserver in the space of 5s *)
END_VAR

VAR
	xAskForTimeOld : BOOL ;
	iSocketIndex : UINT ;
	xBindSocket : BOOL ;
	diTraNr : DINT ;
	udiTime : UDINT ;
	struSOCKADDRESS_Receive : SOCKADDRESS ;
	diRecNr : DINT ;
	diIO : DINT ;
	dwParameterIO : DWORD ;
	arReceiveData : ARRAY[0..3] OF BYTE ;
	xRecIP : BOOL ;
	struInADDR_TimeServer : INADDR;
	striTimeServerIPAddress : STRING;

	TON_Timeout : TON := (PT:=T#5s) ;

	uiRemotePort : UINT := 37 ;
	struSOCKADDRESS_Bind : SOCKADDRESS ;
	struSOCKADDRESS_Transmit : SOCKADDRESS ;
	dwReceiveData : DWORD ;
	udiGMTSecondsSince1970 : UDINT ;
	i : USINT ;

	Split_DT : NetTime_Split_DT ;

	uiDayStartSummertime : UINT ;
	uiDayEndSummertime : UINT ;

	dtStartSummertime : DT ;
	dtEndSummertime : DT ;

	struSOCKADDRESS_Connect : SOCKADDRESS ;
	xSysSockConnect : BOOL ;
END_VAR

IF xActive THEN
	IF NetTime_ar_udiSockets[iSocketIndex] > 0 THEN
		(* waiting for an answer of the time-server *)
		(* is any data received *)
		diIO := SysSockIoctl(NetTime_ar_udiSockets[iSocketIndex], SOCKET_FIONREAD, ADR(dwParameterIO)); (* get num chars available to read *)
		IF dwParameterIO <> 0 THEN
			diRecNr := SysSockRecvFrom(NetTime_ar_udiSockets[iSocketIndex], ADR(arReceiveData), SIZEOF(arReceiveData), 0,
											 ADR(struSOCKADDRESS_Receive), SIZEOF(struSOCKADDRESS_Receive));
			IF diRecNr = -1 THEN
				uiErrorNumber := 4 ;
			ELSE
				(* check receive IP Address *)
				struInADDR_TimeServer.s_addr := struSOCKADDRESS_Receive.sin_addr ;
				xRecIP:=SysSockInetNtoa(struInADDR_TimeServer, striTimeServerIPAddress, SIZEOF(striTimeServerIPAddress)) ;
				IF struSOCKADDRESS_Receive.sin_addr = struSOCKADDRESS_Transmit.sin_addr THEN
					(* answer is coming from requested timeserver *)
					(* interpret received data *)
					(* change byte orientation *)
					dwReceiveData := 0 ;
					FOR i := 0 TO 3 DO
						dwReceiveData := SHL(dwReceiveData,8) ;
						dwReceiveData := dwReceiveData OR BYTE_TO_DWORD(arReceiveData[i]) ;
					END_FOR
					(* dwReceiveData = seconds after 1.1.1900 00:00:00 *)
					IF DWORD_TO_UDINT(dwReceiveData) >= UDINT#2208988800 THEN
						udiGMTSecondsSince1970 := DWORD_TO_UDINT(dwReceiveData) - UDINT#2208988800 ;
					ELSE
						udiGMTSecondsSince1970 := DWORD_TO_UDINT(dwReceiveData) + UDINT#2208988800 ;
					END_IF
					dtReceivedDateTime := UDINT_TO_DT(udiGMTSecondsSince1970+(UINT#3600*SINT_TO_DINT(siGMTOffset))) ;
	
					Split_DT(
						InputDT:=dtReceivedDateTime ,
						uiSecond=>uiReceivedSecond ,
						uiMinute=>uiReceivedMinute ,
						uiHour=>uiReceivedHour ,
						uiDay=>uiReceivedDay ,
						uiMonth=>uiReceivedMonth ,
						uiYear=>uiReceivedYear );
	
					uiReceivedDayOfWeek := NetTime_DayOfWeek(uiReceivedDay,uiReceivedMonth,uiReceivedYear) ;
	
					IF xSummerWinterTime THEN
						(* check if the received time is in summertime interval
						last sunday of march at 2:00 a.m. to last sunday of october at 2:00 a.m. *)
						uiDayStartSummertime := 31-NetTime_DayOfWeek(31,3,uiReceivedYear) ;
						uiDayEndSummertime := 31-NetTime_DayOfWeek(31,10,uiReceivedYear) ;
						dtStartSummertime := NetTime_Concat_DT(0,0,2,uiDayStartSummertime,3,uiReceivedYear) ;
						dtEndSummertime := NetTime_Concat_DT(0,0,2,uiDayEndSummertime,10,uiReceivedYear) ;
						xSummerTime := (dtReceivedDateTime>dtStartSummertime) AND (dtReceivedDateTime<dtEndSummertime) ;
						IF xSummerTime THEN
							(* add 1 hour to GMT time *)
							dtReceivedDateTime := UDINT_TO_DT(DT_TO_UDINT(dtReceivedDateTime) + UDINT#3600) ;
							Split_DT(
								InputDT:=dtReceivedDateTime ,
								uiSecond=>uiReceivedSecond ,
								uiMinute=>uiReceivedMinute ,
								uiHour=>uiReceivedHour ,
								uiDay=>uiReceivedDay ,
								uiMonth=>uiReceivedMonth ,
								uiYear=>uiReceivedYear );
						END_IF
					END_IF
	
					IF xSetRTC THEN
						(* set the local RTC to the received time *)
						SysRtcSetTime(dtReceivedDateTime) ;
					END_IF
	
					(* close socket *)
					NetTime_SockClose(iSocketIndex) ;
					xActive := FALSE ;
				END_IF
			END_IF
	
		ELSE
			TON_Timeout();
			IF TON_Timeout.Q THEN
				uiErrorNumber := 5 ;
				NetTime_SockClose(iSocketIndex) ;
				xActive := FALSE ;
				TON_Timeout(IN:=FALSE) ;
			END_IF
		END_IF
	ELSE
		(* Socketindex is no longer valid! Perhaps PLC has stopt and socket has closed *)
		uiErrorNumber := 5 ;
		xActive := FALSE ;
	END_IF
ELSE
	(* waiting for a new request *)
	IF xAskForTime AND NOT xAskForTimeOld THEN
		(* start time request *)
		dtReceivedDateTime := DATE_AND_TIME#2000-01-01-00:00:00 ;
		uiReceivedSecond := 0 ;
		uiReceivedMinute := 0 ;
		uiReceivedHour := 0 ;
		uiReceivedDay := 1 ;
		uiReceivedMonth := 1 ;
		uiReceivedYear := 2000 ;
		uiReceivedDayOfWeek := 6 ;
		xError := FALSE ;
		uiErrorNumber := 0;
	
		(* create a new  datagram-socket *)
		iSocketIndex := NetTime_SockCreate(SOCKET_AF_INET,SOCKET_DGRAM,0);
		IF iSocketIndex > 0 THEN
			(* Bind the socket to the local port *)
			struSOCKADDRESS_Bind.sin_family := SOCKET_AF_INET; (* internetwork: UDP, TCP, etc. *)
			struSOCKADDRESS_Bind.sin_addr := SysSockHtonl(SOCKET_INADDR_ANY) ;
			struSOCKADDRESS_Bind.sin_port := SysSockHtons(uiLocalPort);
			xBindSocket := SysSockBind(NetTime_ar_udiSockets[iSocketIndex], ADR(struSOCKADDRESS_Bind), SIZEOF(struSOCKADDRESS_Bind));
			IF  xBindSocket THEN
				(* UDP: send a time request to the time server *)
				struSOCKADDRESS_Transmit.sin_family := SOCKET_AF_INET; (* internetwork: UDP, TCP, etc. *)
				struSOCKADDRESS_Transmit.sin_addr := SysSockInetAddr(striIPAddress);
				struSOCKADDRESS_Transmit.sin_port := SysSockHtons(uiRemotePort);
				diTraNr := SysSockSendTo(NetTime_ar_udiSockets[iSocketIndex] , ADR(udiTime), 4,0,
							ADR(struSOCKADDRESS_Transmit), SIZEOF(struSOCKADDRESS_Transmit));
				IF diTraNr < 0 THEN
					uiErrorNumber := 3 ;
					NetTime_SockClose(iSocketIndex) ;
				ELSE
					(* start timeout timer *)
					TON_Timeout(IN:=FALSE) ;
					TON_Timeout(IN:=TRUE) ;
					xActive := TRUE ;
				END_IF
			ELSE
				NetTime_SockClose(iSocketIndex);
				uiErrorNumber := 2 ;
			END_IF
		ELSE
			uiErrorNumber := 1 ;
			NetTime_SockClose(iSocketIndex);
		END_IF
	END_IF
END_IF

xAskForTimeOld := xAskForTime ;
xError := uiErrorNumber<>0 ;

END_FUNCTION_BLOCK

// XV300/Application/POUs/NetTime_RFC868_Client
FUNCTION_BLOCK NetTime_RFC868_Client
(* this FB is a client for time request to a server using a protocol described in RFC868 / UDP *)

VAR_INPUT
	striIPAddress : STRING(15) ; 				(* IP-address of th time server i.e '192.168.0.1' *)
	uiLocalPort : UINT := 1025 ;				(* local ethernet port 1-65535 see RFC1700 for assigned ports *)
	xAskForTime : BOOL ;						(* rising edge send a time request to the server *)
	siGMTOffset : SINT := 1 ;					(* time offset in h for local time-zone (-12..+12) i.e. +1 for Berlin *)
	xSummerWinterTime : BOOL := TRUE ;	(* consider Summertime from last sunday of march at 02:00 a.m.GMT to last sunday of october at 02:00 a.m.GMT *)
	xSetRTC : BOOL ;							(* set the local Real-Time-Clock to the received time from server *)
END_VAR

VAR_OUTPUT
	dtReceivedDateTime : DT := DATE_AND_TIME#2000-01-01-00:00:00 ;		(* received Date and Time from server *)
	uiReceivedSecond : UINT ;				(* received second from server (0..59) *)
	uiReceivedMinute : UINT ;				(* received minute from server (0..59) *)
	uiReceivedHour : UINT ;					(* received hour from server (0..23) *)
	uiReceivedDay : UINT :=1 ;				(* received Day from server (1..31) *)
	uiReceivedMonth : UINT :=1 ;				(* received Month from server (1..12) *)
	uiReceivedYear : UINT :=2000 ;			(* received year from server (2000..2092) *)
	uiReceivedDayOfWeek : UINT := 6 ;		(* received weekday. (1=Monday .. 7=Sunday) *)
	xSummerTime : BOOL ;					(* received Time is Summertime *)
	xActive : BOOL ;							(* waiting for an answer of the time server *)
	xError : BOOL ;							(* last request generate an error - look "uiErrornumber" for reason *)
	uiErrorNumber : UINT ;					(* reason for the last error
		0 = No error
		1 = Ethernet socket could not opend 
		2 = Ethernet socket could not binded
		3 = Transmit time request error
		4 = Ethernet receive error
		5 = Timeout - no answer from timeserver in the space of 5s *)
END_VAR

VAR
	xAskForTimeOld : BOOL ;
	iSocketIndex : UINT ;
	xBindSocket : BOOL ;
	diTraNr : DINT ;
	udiTime : UDINT ;
	struSOCKADDRESS_Receive : SOCKADDRESS ;
	diRecNr : DINT ;
	diIO : DINT ;
	dwParameterIO : DWORD ;
	arReceiveData : ARRAY[0..3] OF BYTE ;
	xRecIP : BOOL ;
	struInADDR_TimeServer : INADDR;
	striTimeServerIPAddress : STRING;

	TON_Timeout : TON := (PT:=T#5s) ;

	uiRemotePort : UINT := 37 ;
	struSOCKADDRESS_Bind : SOCKADDRESS ;
	struSOCKADDRESS_Transmit : SOCKADDRESS ;
	dwReceiveData : DWORD ;
	udiGMTSecondsSince1970 : UDINT ;
	i : USINT ;

	Split_DT : NetTime_Split_DT ;

	uiDayStartSummertime : UINT ;
	uiDayEndSummertime : UINT ;

	dtStartSummertime : DT ;
	dtEndSummertime : DT ;

	struSOCKADDRESS_Connect : SOCKADDRESS ;
	xSysSockConnect : BOOL ;
END_VAR

IF xActive THEN
	IF NetTime_ar_udiSockets[iSocketIndex] > 0 THEN
		(* waiting for an answer of the time-server *)
		(* is any data received *)
		diIO := SysSockIoctl(NetTime_ar_udiSockets[iSocketIndex], SOCKET_FIONREAD, ADR(dwParameterIO)); (* get num chars available to read *)
		IF dwParameterIO <> 0 THEN
			diRecNr := SysSockRecvFrom(NetTime_ar_udiSockets[iSocketIndex], ADR(arReceiveData), SIZEOF(arReceiveData), 0,
											 ADR(struSOCKADDRESS_Receive), SIZEOF(struSOCKADDRESS_Receive));
			IF diRecNr = -1 THEN
				uiErrorNumber := 4 ;
			ELSE
				(* check receive IP Address *)
				struInADDR_TimeServer.s_addr := struSOCKADDRESS_Receive.sin_addr ;
				xRecIP:=SysSockInetNtoa(struInADDR_TimeServer, striTimeServerIPAddress, SIZEOF(striTimeServerIPAddress)) ;
				IF struSOCKADDRESS_Receive.sin_addr = struSOCKADDRESS_Transmit.sin_addr THEN
					(* answer is coming from requested timeserver *)
					(* interpret received data *)
					(* change byte orientation *)
					dwReceiveData := 0 ;
					FOR i := 0 TO 3 DO
						dwReceiveData := SHL(dwReceiveData,8) ;
						dwReceiveData := dwReceiveData OR BYTE_TO_DWORD(arReceiveData[i]) ;
					END_FOR
					(* dwReceiveData = seconds after 1.1.1900 00:00:00 *)
					IF DWORD_TO_UDINT(dwReceiveData) >= UDINT#2208988800 THEN
						udiGMTSecondsSince1970 := DWORD_TO_UDINT(dwReceiveData) - UDINT#2208988800 ;
					ELSE
						udiGMTSecondsSince1970 := DWORD_TO_UDINT(dwReceiveData) + UDINT#2208988800 ;
					END_IF
					dtReceivedDateTime := UDINT_TO_DT(udiGMTSecondsSince1970+(UINT#3600*SINT_TO_DINT(siGMTOffset))) ;
	
					Split_DT(
						InputDT:=dtReceivedDateTime ,
						uiSecond=>uiReceivedSecond ,
						uiMinute=>uiReceivedMinute ,
						uiHour=>uiReceivedHour ,
						uiDay=>uiReceivedDay ,
						uiMonth=>uiReceivedMonth ,
						uiYear=>uiReceivedYear );
	
					uiReceivedDayOfWeek := NetTime_DayOfWeek(uiReceivedDay,uiReceivedMonth,uiReceivedYear) ;
	
					IF xSummerWinterTime THEN
						(* check if the received time is in summertime interval
						last sunday of march at 2:00 a.m. to last sunday of october at 2:00 a.m. *)
						uiDayStartSummertime := 31-NetTime_DayOfWeek(31,3,uiReceivedYear) ;
						uiDayEndSummertime := 31-NetTime_DayOfWeek(31,10,uiReceivedYear) ;
						dtStartSummertime := NetTime_Concat_DT(0,0,2,uiDayStartSummertime,3,uiReceivedYear) ;
						dtEndSummertime := NetTime_Concat_DT(0,0,2,uiDayEndSummertime,10,uiReceivedYear) ;
						xSummerTime := (dtReceivedDateTime>dtStartSummertime) AND (dtReceivedDateTime<dtEndSummertime) ;
						IF xSummerTime THEN
							(* add 1 hour to GMT time *)
							dtReceivedDateTime := UDINT_TO_DT(DT_TO_UDINT(dtReceivedDateTime) + UDINT#3600) ;
							Split_DT(
								InputDT:=dtReceivedDateTime ,
								uiSecond=>uiReceivedSecond ,
								uiMinute=>uiReceivedMinute ,
								uiHour=>uiReceivedHour ,
								uiDay=>uiReceivedDay ,
								uiMonth=>uiReceivedMonth ,
								uiYear=>uiReceivedYear );
						END_IF
					END_IF
	
					IF xSetRTC THEN
						(* set the local RTC to the received time *)
						SysRtcSetTime(dtReceivedDateTime) ;
					END_IF
	
					(* close socket *)
					NetTime_SockClose(iSocketIndex) ;
					xActive := FALSE ;
				END_IF
			END_IF
	
		ELSE
			TON_Timeout();
			IF TON_Timeout.Q THEN
				uiErrorNumber := 5 ;
				NetTime_SockClose(iSocketIndex) ;
				xActive := FALSE ;
				TON_Timeout(IN:=FALSE) ;
			END_IF
		END_IF
	ELSE
		(* Socketindex is no longer valid! Perhaps PLC has stopt and socket has closed *)
		uiErrorNumber := 5 ;
		xActive := FALSE ;
	END_IF
ELSE
	(* waiting for a new request *)
	IF xAskForTime AND NOT xAskForTimeOld THEN
		(* start time request *)
		dtReceivedDateTime := DATE_AND_TIME#2000-01-01-00:00:00 ;
		uiReceivedSecond := 0 ;
		uiReceivedMinute := 0 ;
		uiReceivedHour := 0 ;
		uiReceivedDay := 1 ;
		uiReceivedMonth := 1 ;
		uiReceivedYear := 2000 ;
		uiReceivedDayOfWeek := 6 ;
		xError := FALSE ;
		uiErrorNumber := 0;
	
		(* create a new  datagram-socket *)
		iSocketIndex := NetTime_SockCreate(SOCKET_AF_INET,SOCKET_DGRAM,0);
		IF iSocketIndex > 0 THEN
			(* Bind the socket to the local port *)
			struSOCKADDRESS_Bind.sin_family := SOCKET_AF_INET; (* internetwork: UDP, TCP, etc. *)
			struSOCKADDRESS_Bind.sin_addr := SysSockHtonl(SOCKET_INADDR_ANY) ;
			struSOCKADDRESS_Bind.sin_port := SysSockHtons(uiLocalPort);
			xBindSocket := SysSockBind(NetTime_ar_udiSockets[iSocketIndex], ADR(struSOCKADDRESS_Bind), SIZEOF(struSOCKADDRESS_Bind));
			IF  xBindSocket THEN
				(* UDP: send a time request to the time server *)
				struSOCKADDRESS_Transmit.sin_family := SOCKET_AF_INET; (* internetwork: UDP, TCP, etc. *)
				struSOCKADDRESS_Transmit.sin_addr := SysSockInetAddr(striIPAddress);
				struSOCKADDRESS_Transmit.sin_port := SysSockHtons(uiRemotePort);
				diTraNr := SysSockSendTo(NetTime_ar_udiSockets[iSocketIndex] , ADR(udiTime), 4,0,
							ADR(struSOCKADDRESS_Transmit), SIZEOF(struSOCKADDRESS_Transmit));
				IF diTraNr < 0 THEN
					uiErrorNumber := 3 ;
					NetTime_SockClose(iSocketIndex) ;
				ELSE
					(* start timeout timer *)
					TON_Timeout(IN:=FALSE) ;
					TON_Timeout(IN:=TRUE) ;
					xActive := TRUE ;
				END_IF
			ELSE
				NetTime_SockClose(iSocketIndex);
				uiErrorNumber := 2 ;
			END_IF
		ELSE
			uiErrorNumber := 1 ;
			NetTime_SockClose(iSocketIndex);
		END_IF
	END_IF
END_IF

xAskForTimeOld := xAskForTime ;
xError := uiErrorNumber<>0 ;

END_FUNCTION_BLOCK

// XC303/Application/POUs/Internal/NetTime_Split_DT
FUNCTION_BLOCK NetTime_Split_DT
(* Split datatype Date_And_Time *)

VAR_INPUT
	InputDT : DT;
END_VAR
VAR_OUTPUT
	uiSecond : UINT ;
	uiMinute : UINT ;
	uiHour : UINT ;
	uiDay : UINT ;
	uiMonth : UINT ;
	uiYear : UINT ;
END_VAR

VAR
	Error			: BOOL;
	dw_date_g					: DWORD;
	dw_date_rest					: DWORD;
	dw_date_y						: DWORD;
	dw_leap_block				: DWORD;
	dw_day_g						: DWORD;
	dw_year_number				: DWORD;
	dw_leapblocks_seconds		: DWORD;
	dw_day_leap_g				: DWORD;
	dw_day_month				: DWORD;
	dw_year_offset_seconds		: DWORD;
	dw_time_rest					: DWORD;
	dw_hours						: DWORD;
	dw_minuts					: DWORD;
END_VAR
VAR CONSTANT
	dw_day_seconds				: DWORD:=86400;
	dw_year_seconds			: DWORD:=31536000;
	dw_offset_seconds_73		: DWORD:=94694400;
	dw_leapblock_seconds		: DWORD:=126230400;
END_VAR

// NETWORK 1
// instruction list
LD      0
ST      error

// NETWORK 2
// instruction list
LD      InputDT
DT_TO_DWORD
SUB     dw_offset_seconds_73
ST      dw_date_g

// NETWORK 3
// instruction list
LD      dw_date_g
DIV     dw_leapblock_seconds
ST      dw_leap_block

// NETWORK 4
// instruction list
LD      dw_leap_block
MUL     dw_leapblock_seconds
ST      dw_leapblocks_seconds

// NETWORK 5
// instruction list
LD      dw_date_g
MOD     dw_leapblocks_seconds
ST      dw_date_rest

// NETWORK 6
// instruction list
LD      dw_leap_block
MUL     4
ST      dw_date_y

// NETWORK 7
// instruction list
LD      0
ST      dw_year_number

// NETWORK 8
// instruction list
LD      dw_date_rest
EQ      0
JMPC    set_year

// NETWORK 9
// instruction list
LD      dw_date_rest
DIV     dw_year_seconds
ST      dw_year_number

// NETWORK 10
// instruction list
LD      dw_year_number
GT      3
JMPCN   set_year

// NETWORK 11
// instruction list
LD      dw_year_number
SUB     1
ST      dw_year_number

// NETWORK 12
set_year:
// instruction list
LD      dw_year_number
ADD     dw_date_y
DWORD_TO_UINT
ADD     1973
ST      uiYear

// NETWORK 13
// instruction list
LD      uiYear
LT      1993
JMPC    error

// NETWORK 14
// instruction list
LD      uiYear
GT      2092
JMPC    error

// NETWORK 15
get_month:
// instruction list
LD      dw_year_number
MUL     dw_year_seconds
ST      dw_year_offset_seconds

// NETWORK 16
// instruction list
LD      dw_date_rest
SUB     dw_year_offset_seconds
DIV     dw_day_seconds
ADD     1
ST      dw_day_g
ST      dw_day_leap_g

// NETWORK 17
jan:
// instruction list
LD      dw_day_g
GT      31
JMPC    feb

// NETWORK 18
// instruction list
LD      1
ST      uiMonth

// NETWORK 19
// instruction list
LD      dw_day_g
ST      dw_day_month
JMP     get_days

// NETWORK 20
feb:
// instruction list
LD      dw_day_g
GT      60
JMPC    verify_leap_year

// NETWORK 21
// instruction list
LD      dw_year_number
EQ      3
JMPC    set_feb

// NETWORK 22
// instruction list
LD      dw_day_g
EQ      60
JMPC    mar

// NETWORK 23
set_feb:
// instruction list
LD      2
ST      uiMonth

// NETWORK 24
// instruction list
LD      dw_day_g
SUB     31
ST      dw_day_month
JMP     get_days

// NETWORK 25
verify_leap_year:
// instruction list
LD      dw_year_number
EQ      3
JMPCN   mar

// NETWORK 26
// instruction list
LD      dw_day_g
SUB     1
ST      dw_day_leap_g

// NETWORK 27
mar:
// instruction list
LD      dw_day_leap_g
GT      90
JMPC    apr

// NETWORK 28
// instruction list
LD      3
ST      uiMonth

// NETWORK 29
// instruction list
LD      dw_day_leap_g
SUB     59
ST      dw_day_month
JMP     get_days

// NETWORK 30
apr:
// instruction list
LD      dw_day_leap_g
GT      120
JMPC    may

// NETWORK 31
// instruction list
LD      4
ST      uiMonth

// NETWORK 32
// instruction list
LD      dw_day_leap_g
SUB     90
ST      dw_day_month
JMP     get_days

// NETWORK 33
may:
// instruction list
LD      dw_day_leap_g
GT      151
JMPC    jun

// NETWORK 34
// instruction list
LD      5
ST      uiMonth

// NETWORK 35
// instruction list
LD      dw_day_leap_g
SUB     120
ST      dw_day_month
JMP     get_days

// NETWORK 36
jun:
// instruction list
LD      dw_day_leap_g
GT      181
JMPC    jul

// NETWORK 37
// instruction list
LD      6
ST      uiMonth

// NETWORK 38
// instruction list
LD      dw_day_leap_g
SUB     151
ST      dw_day_month
JMP     get_days

// NETWORK 39
jul:
// instruction list
LD      dw_day_leap_g
GT      212
JMPC    aug

// NETWORK 40
// instruction list
LD      7
ST      uiMonth

// NETWORK 41
// instruction list
LD      dw_day_leap_g
SUB     181
ST      dw_day_month
JMP     get_days

// NETWORK 42
aug:
// instruction list
LD      dw_day_leap_g
GT      243
JMPC    sep

// NETWORK 43
// instruction list
LD      8
ST      uiMonth

// NETWORK 44
// instruction list
LD      dw_day_leap_g
SUB     212
ST      dw_day_month
JMP     get_days

// NETWORK 45
sep:
// instruction list
LD      dw_day_leap_g
GT      273
JMPC    okt

// NETWORK 46
// instruction list
LD      9
ST      uiMonth

// NETWORK 47
// instruction list
LD      dw_day_leap_g
SUB     243
ST      dw_day_month
JMP     get_days

// NETWORK 48
okt:
// instruction list
LD      dw_day_leap_g
GT      304
JMPC    nov

// NETWORK 49
// instruction list
LD      10
ST      uiMonth

// NETWORK 50
// instruction list
LD      dw_day_leap_g
SUB     273
ST      dw_day_month
JMP     get_days

// NETWORK 51
nov:
// instruction list
LD      dw_day_leap_g
GT      334
JMPC    dez

// NETWORK 52
// instruction list
LD      11
ST      uiMonth

// NETWORK 53
// instruction list
LD      dw_day_leap_g
SUB     304
ST      dw_day_month
JMP     get_days

// NETWORK 54
dez:
// instruction list
LD      dw_day_leap_g
GT      365
JMPC    error

// NETWORK 55
// instruction list
LD      12
ST      uiMonth

// NETWORK 56
// instruction list
LD      dw_day_leap_g
SUB     334
ST      dw_day_month
JMP     get_days

// NETWORK 57
get_days:
// instruction list
LD      dw_day_month
DWORD_TO_UINT
ST      uiDay

// NETWORK 58
get_time:
// instruction list
LD      dw_date_rest
MOD     dw_day_seconds
ST      dw_time_rest

// NETWORK 59
get_hour:
// instruction list
LD      dw_time_rest
DIV     3600
ST      dw_hours

// NETWORK 60
// instruction list
LD      dw_hours
DWORD_TO_UINT
ST      uiHour

// NETWORK 61
// instruction list
LD      dw_time_rest
MOD     3600
ST      dw_time_rest

// NETWORK 62
get_minute:
// instruction list
LD      dw_time_rest
DIV     60
ST      dw_minuts

// NETWORK 63
// instruction list
LD      dw_minuts
DWORD_TO_UINT
ST      uiMinute

// NETWORK 64
// instruction list
LD      dw_time_rest
MOD     60
ST      dw_time_rest

// NETWORK 65
get_sekunde:
// instruction list
LD      dw_time_rest
DWORD_TO_UINT
ST      uiSecond
JMP     ende

// NETWORK 66
error:
// instruction list
LD      1
ST      error

// NETWORK 67
// instruction list
LD      59
ST      uiSecond
ST      uiMinute

// NETWORK 68
// instruction list
LD      23
ST      uiHour

// NETWORK 69
// instruction list
LD      31
ST      uiDay

// NETWORK 70
// instruction list
LD      12
ST      uiMonth

// NETWORK 71
// instruction list
LD      1993
ST      uiYear

// NETWORK 72
ende:
// instruction list

END_FUNCTION_BLOCK

// XV100/Application/POUs/Internal/NetTime_Split_DT
FUNCTION_BLOCK NetTime_Split_DT
(* Split datatype Date_And_Time *)

VAR_INPUT
	InputDT : DT;
END_VAR
VAR_OUTPUT
	uiSecond : UINT ;
	uiMinute : UINT ;
	uiHour : UINT ;
	uiDay : UINT ;
	uiMonth : UINT ;
	uiYear : UINT ;
END_VAR

VAR
	Error			: BOOL;
	dw_date_g					: DWORD;
	dw_date_rest					: DWORD;
	dw_date_y						: DWORD;
	dw_leap_block				: DWORD;
	dw_day_g						: DWORD;
	dw_year_number				: DWORD;
	dw_leapblocks_seconds		: DWORD;
	dw_day_leap_g				: DWORD;
	dw_day_month				: DWORD;
	dw_year_offset_seconds		: DWORD;
	dw_time_rest					: DWORD;
	dw_hours						: DWORD;
	dw_minuts					: DWORD;
END_VAR
VAR CONSTANT
	dw_day_seconds				: DWORD:=86400;
	dw_year_seconds			: DWORD:=31536000;
	dw_offset_seconds_73		: DWORD:=94694400;
	dw_leapblock_seconds		: DWORD:=126230400;
END_VAR

// NETWORK 1
// instruction list
LD      0
ST      error

// NETWORK 2
// instruction list
LD      InputDT
DT_TO_DWORD
SUB     dw_offset_seconds_73
ST      dw_date_g

// NETWORK 3
// instruction list
LD      dw_date_g
DIV     dw_leapblock_seconds
ST      dw_leap_block

// NETWORK 4
// instruction list
LD      dw_leap_block
MUL     dw_leapblock_seconds
ST      dw_leapblocks_seconds

// NETWORK 5
// instruction list
LD      dw_date_g
MOD     dw_leapblocks_seconds
ST      dw_date_rest

// NETWORK 6
// instruction list
LD      dw_leap_block
MUL     4
ST      dw_date_y

// NETWORK 7
// instruction list
LD      0
ST      dw_year_number

// NETWORK 8
// instruction list
LD      dw_date_rest
EQ      0
JMPC    set_year

// NETWORK 9
// instruction list
LD      dw_date_rest
DIV     dw_year_seconds
ST      dw_year_number

// NETWORK 10
// instruction list
LD      dw_year_number
GT      3
JMPCN   set_year

// NETWORK 11
// instruction list
LD      dw_year_number
SUB     1
ST      dw_year_number

// NETWORK 12
set_year:
// instruction list
LD      dw_year_number
ADD     dw_date_y
DWORD_TO_UINT
ADD     1973
ST      uiYear

// NETWORK 13
// instruction list
LD      uiYear
LT      1993
JMPC    error

// NETWORK 14
// instruction list
LD      uiYear
GT      2092
JMPC    error

// NETWORK 15
get_month:
// instruction list
LD      dw_year_number
MUL     dw_year_seconds
ST      dw_year_offset_seconds

// NETWORK 16
// instruction list
LD      dw_date_rest
SUB     dw_year_offset_seconds
DIV     dw_day_seconds
ADD     1
ST      dw_day_g
ST      dw_day_leap_g

// NETWORK 17
jan:
// instruction list
LD      dw_day_g
GT      31
JMPC    feb

// NETWORK 18
// instruction list
LD      1
ST      uiMonth

// NETWORK 19
// instruction list
LD      dw_day_g
ST      dw_day_month
JMP     get_days

// NETWORK 20
feb:
// instruction list
LD      dw_day_g
GT      60
JMPC    verify_leap_year

// NETWORK 21
// instruction list
LD      dw_year_number
EQ      3
JMPC    set_feb

// NETWORK 22
// instruction list
LD      dw_day_g
EQ      60
JMPC    mar

// NETWORK 23
set_feb:
// instruction list
LD      2
ST      uiMonth

// NETWORK 24
// instruction list
LD      dw_day_g
SUB     31
ST      dw_day_month
JMP     get_days

// NETWORK 25
verify_leap_year:
// instruction list
LD      dw_year_number
EQ      3
JMPCN   mar

// NETWORK 26
// instruction list
LD      dw_day_g
SUB     1
ST      dw_day_leap_g

// NETWORK 27
mar:
// instruction list
LD      dw_day_leap_g
GT      90
JMPC    apr

// NETWORK 28
// instruction list
LD      3
ST      uiMonth

// NETWORK 29
// instruction list
LD      dw_day_leap_g
SUB     59
ST      dw_day_month
JMP     get_days

// NETWORK 30
apr:
// instruction list
LD      dw_day_leap_g
GT      120
JMPC    may

// NETWORK 31
// instruction list
LD      4
ST      uiMonth

// NETWORK 32
// instruction list
LD      dw_day_leap_g
SUB     90
ST      dw_day_month
JMP     get_days

// NETWORK 33
may:
// instruction list
LD      dw_day_leap_g
GT      151
JMPC    jun

// NETWORK 34
// instruction list
LD      5
ST      uiMonth

// NETWORK 35
// instruction list
LD      dw_day_leap_g
SUB     120
ST      dw_day_month
JMP     get_days

// NETWORK 36
jun:
// instruction list
LD      dw_day_leap_g
GT      181
JMPC    jul

// NETWORK 37
// instruction list
LD      6
ST      uiMonth

// NETWORK 38
// instruction list
LD      dw_day_leap_g
SUB     151
ST      dw_day_month
JMP     get_days

// NETWORK 39
jul:
// instruction list
LD      dw_day_leap_g
GT      212
JMPC    aug

// NETWORK 40
// instruction list
LD      7
ST      uiMonth

// NETWORK 41
// instruction list
LD      dw_day_leap_g
SUB     181
ST      dw_day_month
JMP     get_days

// NETWORK 42
aug:
// instruction list
LD      dw_day_leap_g
GT      243
JMPC    sep

// NETWORK 43
// instruction list
LD      8
ST      uiMonth

// NETWORK 44
// instruction list
LD      dw_day_leap_g
SUB     212
ST      dw_day_month
JMP     get_days

// NETWORK 45
sep:
// instruction list
LD      dw_day_leap_g
GT      273
JMPC    okt

// NETWORK 46
// instruction list
LD      9
ST      uiMonth

// NETWORK 47
// instruction list
LD      dw_day_leap_g
SUB     243
ST      dw_day_month
JMP     get_days

// NETWORK 48
okt:
// instruction list
LD      dw_day_leap_g
GT      304
JMPC    nov

// NETWORK 49
// instruction list
LD      10
ST      uiMonth

// NETWORK 50
// instruction list
LD      dw_day_leap_g
SUB     273
ST      dw_day_month
JMP     get_days

// NETWORK 51
nov:
// instruction list
LD      dw_day_leap_g
GT      334
JMPC    dez

// NETWORK 52
// instruction list
LD      11
ST      uiMonth

// NETWORK 53
// instruction list
LD      dw_day_leap_g
SUB     304
ST      dw_day_month
JMP     get_days

// NETWORK 54
dez:
// instruction list
LD      dw_day_leap_g
GT      365
JMPC    error

// NETWORK 55
// instruction list
LD      12
ST      uiMonth

// NETWORK 56
// instruction list
LD      dw_day_leap_g
SUB     334
ST      dw_day_month
JMP     get_days

// NETWORK 57
get_days:
// instruction list
LD      dw_day_month
DWORD_TO_UINT
ST      uiDay

// NETWORK 58
get_time:
// instruction list
LD      dw_date_rest
MOD     dw_day_seconds
ST      dw_time_rest

// NETWORK 59
get_hour:
// instruction list
LD      dw_time_rest
DIV     3600
ST      dw_hours

// NETWORK 60
// instruction list
LD      dw_hours
DWORD_TO_UINT
ST      uiHour

// NETWORK 61
// instruction list
LD      dw_time_rest
MOD     3600
ST      dw_time_rest

// NETWORK 62
get_minute:
// instruction list
LD      dw_time_rest
DIV     60
ST      dw_minuts

// NETWORK 63
// instruction list
LD      dw_minuts
DWORD_TO_UINT
ST      uiMinute

// NETWORK 64
// instruction list
LD      dw_time_rest
MOD     60
ST      dw_time_rest

// NETWORK 65
get_sekunde:
// instruction list
LD      dw_time_rest
DWORD_TO_UINT
ST      uiSecond
JMP     ende

// NETWORK 66
error:
// instruction list
LD      1
ST      error

// NETWORK 67
// instruction list
LD      59
ST      uiSecond
ST      uiMinute

// NETWORK 68
// instruction list
LD      23
ST      uiHour

// NETWORK 69
// instruction list
LD      31
ST      uiDay

// NETWORK 70
// instruction list
LD      12
ST      uiMonth

// NETWORK 71
// instruction list
LD      1993
ST      uiYear

// NETWORK 72
ende:
// instruction list

END_FUNCTION_BLOCK

// XV300/Application/POUs/Internal/NetTime_Split_DT
FUNCTION_BLOCK NetTime_Split_DT
(* Split datatype Date_And_Time *)

VAR_INPUT
	InputDT : DT;
END_VAR
VAR_OUTPUT
	uiSecond : UINT ;
	uiMinute : UINT ;
	uiHour : UINT ;
	uiDay : UINT ;
	uiMonth : UINT ;
	uiYear : UINT ;
END_VAR

VAR
	Error			: BOOL;
	dw_date_g					: DWORD;
	dw_date_rest					: DWORD;
	dw_date_y						: DWORD;
	dw_leap_block				: DWORD;
	dw_day_g						: DWORD;
	dw_year_number				: DWORD;
	dw_leapblocks_seconds		: DWORD;
	dw_day_leap_g				: DWORD;
	dw_day_month				: DWORD;
	dw_year_offset_seconds		: DWORD;
	dw_time_rest					: DWORD;
	dw_hours						: DWORD;
	dw_minuts					: DWORD;
END_VAR
VAR CONSTANT
	dw_day_seconds				: DWORD:=86400;
	dw_year_seconds			: DWORD:=31536000;
	dw_offset_seconds_73		: DWORD:=94694400;
	dw_leapblock_seconds		: DWORD:=126230400;
END_VAR

// NETWORK 1
// instruction list
LD      0
ST      error

// NETWORK 2
// instruction list
LD      InputDT
DT_TO_DWORD
SUB     dw_offset_seconds_73
ST      dw_date_g

// NETWORK 3
// instruction list
LD      dw_date_g
DIV     dw_leapblock_seconds
ST      dw_leap_block

// NETWORK 4
// instruction list
LD      dw_leap_block
MUL     dw_leapblock_seconds
ST      dw_leapblocks_seconds

// NETWORK 5
// instruction list
LD      dw_date_g
MOD     dw_leapblocks_seconds
ST      dw_date_rest

// NETWORK 6
// instruction list
LD      dw_leap_block
MUL     4
ST      dw_date_y

// NETWORK 7
// instruction list
LD      0
ST      dw_year_number

// NETWORK 8
// instruction list
LD      dw_date_rest
EQ      0
JMPC    set_year

// NETWORK 9
// instruction list
LD      dw_date_rest
DIV     dw_year_seconds
ST      dw_year_number

// NETWORK 10
// instruction list
LD      dw_year_number
GT      3
JMPCN   set_year

// NETWORK 11
// instruction list
LD      dw_year_number
SUB     1
ST      dw_year_number

// NETWORK 12
set_year:
// instruction list
LD      dw_year_number
ADD     dw_date_y
DWORD_TO_UINT
ADD     1973
ST      uiYear

// NETWORK 13
// instruction list
LD      uiYear
LT      1993
JMPC    error

// NETWORK 14
// instruction list
LD      uiYear
GT      2092
JMPC    error

// NETWORK 15
get_month:
// instruction list
LD      dw_year_number
MUL     dw_year_seconds
ST      dw_year_offset_seconds

// NETWORK 16
// instruction list
LD      dw_date_rest
SUB     dw_year_offset_seconds
DIV     dw_day_seconds
ADD     1
ST      dw_day_g
ST      dw_day_leap_g

// NETWORK 17
jan:
// instruction list
LD      dw_day_g
GT      31
JMPC    feb

// NETWORK 18
// instruction list
LD      1
ST      uiMonth

// NETWORK 19
// instruction list
LD      dw_day_g
ST      dw_day_month
JMP     get_days

// NETWORK 20
feb:
// instruction list
LD      dw_day_g
GT      60
JMPC    verify_leap_year

// NETWORK 21
// instruction list
LD      dw_year_number
EQ      3
JMPC    set_feb

// NETWORK 22
// instruction list
LD      dw_day_g
EQ      60
JMPC    mar

// NETWORK 23
set_feb:
// instruction list
LD      2
ST      uiMonth

// NETWORK 24
// instruction list
LD      dw_day_g
SUB     31
ST      dw_day_month
JMP     get_days

// NETWORK 25
verify_leap_year:
// instruction list
LD      dw_year_number
EQ      3
JMPCN   mar

// NETWORK 26
// instruction list
LD      dw_day_g
SUB     1
ST      dw_day_leap_g

// NETWORK 27
mar:
// instruction list
LD      dw_day_leap_g
GT      90
JMPC    apr

// NETWORK 28
// instruction list
LD      3
ST      uiMonth

// NETWORK 29
// instruction list
LD      dw_day_leap_g
SUB     59
ST      dw_day_month
JMP     get_days

// NETWORK 30
apr:
// instruction list
LD      dw_day_leap_g
GT      120
JMPC    may

// NETWORK 31
// instruction list
LD      4
ST      uiMonth

// NETWORK 32
// instruction list
LD      dw_day_leap_g
SUB     90
ST      dw_day_month
JMP     get_days

// NETWORK 33
may:
// instruction list
LD      dw_day_leap_g
GT      151
JMPC    jun

// NETWORK 34
// instruction list
LD      5
ST      uiMonth

// NETWORK 35
// instruction list
LD      dw_day_leap_g
SUB     120
ST      dw_day_month
JMP     get_days

// NETWORK 36
jun:
// instruction list
LD      dw_day_leap_g
GT      181
JMPC    jul

// NETWORK 37
// instruction list
LD      6
ST      uiMonth

// NETWORK 38
// instruction list
LD      dw_day_leap_g
SUB     151
ST      dw_day_month
JMP     get_days

// NETWORK 39
jul:
// instruction list
LD      dw_day_leap_g
GT      212
JMPC    aug

// NETWORK 40
// instruction list
LD      7
ST      uiMonth

// NETWORK 41
// instruction list
LD      dw_day_leap_g
SUB     181
ST      dw_day_month
JMP     get_days

// NETWORK 42
aug:
// instruction list
LD      dw_day_leap_g
GT      243
JMPC    sep

// NETWORK 43
// instruction list
LD      8
ST      uiMonth

// NETWORK 44
// instruction list
LD      dw_day_leap_g
SUB     212
ST      dw_day_month
JMP     get_days

// NETWORK 45
sep:
// instruction list
LD      dw_day_leap_g
GT      273
JMPC    okt

// NETWORK 46
// instruction list
LD      9
ST      uiMonth

// NETWORK 47
// instruction list
LD      dw_day_leap_g
SUB     243
ST      dw_day_month
JMP     get_days

// NETWORK 48
okt:
// instruction list
LD      dw_day_leap_g
GT      304
JMPC    nov

// NETWORK 49
// instruction list
LD      10
ST      uiMonth

// NETWORK 50
// instruction list
LD      dw_day_leap_g
SUB     273
ST      dw_day_month
JMP     get_days

// NETWORK 51
nov:
// instruction list
LD      dw_day_leap_g
GT      334
JMPC    dez

// NETWORK 52
// instruction list
LD      11
ST      uiMonth

// NETWORK 53
// instruction list
LD      dw_day_leap_g
SUB     304
ST      dw_day_month
JMP     get_days

// NETWORK 54
dez:
// instruction list
LD      dw_day_leap_g
GT      365
JMPC    error

// NETWORK 55
// instruction list
LD      12
ST      uiMonth

// NETWORK 56
// instruction list
LD      dw_day_leap_g
SUB     334
ST      dw_day_month
JMP     get_days

// NETWORK 57
get_days:
// instruction list
LD      dw_day_month
DWORD_TO_UINT
ST      uiDay

// NETWORK 58
get_time:
// instruction list
LD      dw_date_rest
MOD     dw_day_seconds
ST      dw_time_rest

// NETWORK 59
get_hour:
// instruction list
LD      dw_time_rest
DIV     3600
ST      dw_hours

// NETWORK 60
// instruction list
LD      dw_hours
DWORD_TO_UINT
ST      uiHour

// NETWORK 61
// instruction list
LD      dw_time_rest
MOD     3600
ST      dw_time_rest

// NETWORK 62
get_minute:
// instruction list
LD      dw_time_rest
DIV     60
ST      dw_minuts

// NETWORK 63
// instruction list
LD      dw_minuts
DWORD_TO_UINT
ST      uiMinute

// NETWORK 64
// instruction list
LD      dw_time_rest
MOD     60
ST      dw_time_rest

// NETWORK 65
get_sekunde:
// instruction list
LD      dw_time_rest
DWORD_TO_UINT
ST      uiSecond
JMP     ende

// NETWORK 66
error:
// instruction list
LD      1
ST      error

// NETWORK 67
// instruction list
LD      59
ST      uiSecond
ST      uiMinute

// NETWORK 68
// instruction list
LD      23
ST      uiHour

// NETWORK 69
// instruction list
LD      31
ST      uiDay

// NETWORK 70
// instruction list
LD      12
ST      uiMonth

// NETWORK 71
// instruction list
LD      1993
ST      uiYear

// NETWORK 72
ende:
// instruction list

END_FUNCTION_BLOCK

// XC303/Application/POUs/NetTime_RFC868_Server
FUNCTION_BLOCK NetTime_RFC868_Server (* prefix: srv868 *)
(* this FB is a server for time request from a client using a protocol described in RFC868 UDP *)
VAR_INPUT
	xEnable : BOOL ;							(* TRUE enable the server if there are no error, FALSE stop it and reset error *)
	siGMTOffset : SINT := 1 ;					(* time offset in h for local time-zone (-12..+12) i.e. +1 for Berlin *)
	xSummerWinterTime : BOOL := TRUE  ;	(* consider Summertime from last sunday of march at 02:00 a.m.GMT to last sunday of october at 02:00 a.m.GMT *)
END_VAR

VAR_OUTPUT
	xActive : BOOL ;							(* server active, waiting for an request *)
	uiCountOfRequest : UINT ;				(* count of requests from a client *)
	sTimeClientIPAddress : STRING ;	(* IP address of the last client request *)
	xError : BOOL ;							(* last start or request generate an error - look "uiErrornumber" for reason *)
	uiErrorNumber : UINT ;					(* reason for the last error
		0 = No error
		1 = Ethernet socket could not opend 
		2 = Ethernet socket could not binded
		3 = Transmit time answer error
		4 = Ethernet receive error *)
END_VAR

VAR
	iSocketIndex : INT ;
	xBindSocket : BOOL ;

	diTraNr : DINT ;

	struSOCKADDRESS_Client : SOCKADDRESS ;
	diRecNr : DINT ;
	diIO : DINT ;
	dwParameterIO : DWORD ;
	arReceiveData : ARRAY[0..3] OF BYTE ;
	xSockInetNtoa : BOOL ;
	struInADDR_Client : INADDR;
	struSOCKADDRESS_Local : SOCKADDRESS ;
	uiLocalPort : UINT := 37 ;


	dtDateTime : DT ;
	uiSecond : UINT ;
	uiMinute : UINT ;
	uiHour : UINT ;
	uiDay : UINT ;
	uiMonth : UINT ;
	uiYear :UINT ;
	uiDayOfWeek : UINT ;
	xSummerTime : BOOL ;

	i : USINT ;

	Split_DT : NetTime_Split_DT ;

	uiDayStartSummertime : UINT ;
	uiDayEndSummertime : UINT ;
	dtStartSummertime : DT ;
	dtEndSummertime : DT ;

	udiGMTSecondsSince1900 : UDINT ;
	ptrSendData : POINTER TO ARRAY[0..3] OF BYTE ;
	arSendData : ARRAY[0..3] OF BYTE ;
	dwSendData : DWORD ;


END_VAR

IF xActive THEN
	IF xEnable THEN
		IF NetTime_ar_udiSockets[iSocketIndex] > 0 THEN
			(* waiting for an request.  Is any data received? *)
			diIO := SysSockIoctl(NetTime_ar_udiSockets[iSocketIndex], SOCKET_FIONREAD, ADR(dwParameterIO)); (* get num chars available to read *)
			IF dwParameterIO <> 0 THEN
				diRecNr := SysSockRecvFrom(NetTime_ar_udiSockets[iSocketIndex], ADR(arReceiveData), SIZEOF(arReceiveData), 0,
												 ADR(struSOCKADDRESS_Client), SIZEOF(struSOCKADDRESS_Client));
				IF diRecNr = -1 THEN
					uiErrorNumber := 4 ;
					xActive := FALSE ;
					NetTime_SockClose(iSocketIndex) ;
				ELSE
					uiCountOfRequest := uiCountOfRequest + 1 ;
					(* check receive IP Address *)
					struInADDR_Client.s_addr := struSOCKADDRESS_Client.sin_addr ;
					xSockInetNtoa:=SysSockInetNtoa(struInADDR_Client, sTimeClientIPAddress, SIZEOF(sTimeClientIPAddress)) ;

					(* get local real time clock *)
					dtDateTime :=SysRtcGetTime(TRUE) ;

					(* sub GMTOffset to get GMT *)
					dtDateTime := UDINT_TO_DT(DT_TO_UDINT(dtDateTime)-(DINT#3600*SINT_TO_DINT(siGMTOffset))) ;

					Split_DT(
						InputDT:=dtDateTime ,
						uiSecond=>uiSecond ,
						uiMinute=>uiMinute ,
						uiHour=>uiHour ,
						uiDay=>uiDay ,
						uiMonth=>uiMonth ,
						uiYear=>uiYear );

					uiDayOfWeek := NetTime_DayOfWeek(uiDay,uiMonth,uiYear) ;

					IF xSummerWinterTime THEN
						(* check if the actual time is in summertime interval
						last sunday of march at 2:00 a.m. to last sunday of october at 2:00 a.m. *)
						uiDayStartSummertime := 31-NetTime_DayOfWeek(31,3,uiYear) ;
						uiDayEndSummertime := 31-NetTime_DayOfWeek(31,10,uiYear) ;
						dtStartSummertime := NetTime_Concat_DT(0,0,2,uiDayStartSummertime,3,uiYear) ;
						dtEndSummertime := NetTime_Concat_DT(0,0,2,uiDayEndSummertime,10,uiYear) ;
						xSummerTime := (dtDateTime>dtStartSummertime) AND (dtDateTime<dtEndSummertime) ;
						IF xSummerTime THEN
							(* sub 1 hour to get GMT time *)
							dtDateTime := UDINT_TO_DT(DT_TO_UDINT(dtDateTime) - UDINT#3600) ;
							Split_DT(
								InputDT:=dtDateTime ,
								uiSecond=>uiSecond ,
								uiMinute=>uiMinute ,
								uiHour=>uiHour ,
								uiDay=>uiDay ,
								uiMonth=>uiMonth ,
								uiYear=>uiYear );
						END_IF
					END_IF

					udiGMTSecondsSince1900 := DT_TO_UDINT(dtDateTime) + UDINT#2208988800 ;

					ptrSendData := ADR(udiGMTSecondsSince1900) ;
					arSendData := ptrSendData^ ;

					(* change byte orientation *)
					dwSendData := 0 ;
					FOR i := 0 TO 3 DO
						dwSendData := SHL(dwSendData,8) ;
						dwSendData := dwSendData OR BYTE_TO_DWORD(arSendData[i]) ;
					END_FOR

					diTraNr := SysSockSendTo(NetTime_ar_udiSockets[iSocketIndex] , ADR(dwSendData), 4,0,
								ADR(struSOCKADDRESS_Client), SIZEOF(struSOCKADDRESS_Client));
					IF diTraNr < 0 THEN
						uiErrorNumber := 3 ;
						xActive := FALSE ;
						NetTime_SockClose(iSocketIndex) ;
					END_IF
				END_IF
			END_IF
		ELSE
			(* Socketindex is no longer valid! Perhaps PLC has stopt and socket has closed *)
			xActive := FALSE ;
			uiCountOfRequest := 0 ;
			sTimeClientIPAddress := '' ;
			xError := FALSE ;
			uiErrorNumber := 0 ;
		END_IF
	ELSE
		(* stop time server *)
		NetTime_SockClose(iSocketIndex) ;
		xActive := FALSE ;
		uiCountOfRequest := 0 ;
		sTimeClientIPAddress := '' ;
		xError := FALSE ;
		uiErrorNumber := 0 ;
	END_IF
ELSE
	IF xEnable THEN
		IF NOT xError THEN
			(* start timeserver *)
			xError := FALSE ;
			uiErrorNumber := 0;

			(* create a new  datagram-socket *)
			iSocketIndex := NetTime_SockCreate(SOCKET_AF_INET,SOCKET_DGRAM,0);
			IF iSocketIndex > 0 THEN
				(* Bind the socket to the local port *)
				struSOCKADDRESS_Local.sin_family := SOCKET_AF_INET; (* internetwork: UDP, TCP, etc. *)
				struSOCKADDRESS_Local.sin_addr := SysSockHtonl(SOCKET_INADDR_ANY) ;
				struSOCKADDRESS_Local.sin_port := SysSockHtons(uiLocalPort);
				xBindSocket := SysSockBind(NetTime_ar_udiSockets[iSocketIndex], ADR(struSOCKADDRESS_Local), SIZEOF(struSOCKADDRESS_Local));
				IF  NOT xBindSocket THEN
					NetTime_SockClose(iSocketIndex);
					uiErrorNumber := 2 ;
				ELSE
					xActive := TRUE ;
				END_IF
			ELSE
				uiErrorNumber := 1 ;
				NetTime_SockClose(iSocketIndex);
			END_IF
		END_IF
	ELSE
		(* reset last error *)
		uiCountOfRequest := 0 ;
		sTimeClientIPAddress := '' ;
		xError := FALSE ;
		uiErrorNumber := 0 ;
	END_IF
END_IF

xError := uiErrorNumber<>0 ;

END_FUNCTION_BLOCK

// XV100/Application/POUs/NetTime_RFC868_Server
FUNCTION_BLOCK NetTime_RFC868_Server (* prefix: srv868 *)
(* this FB is a server for time request from a client using a protocol described in RFC868 UDP *)
VAR_INPUT
	xEnable : BOOL ;							(* TRUE enable the server if there are no error, FALSE stop it and reset error *)
	siGMTOffset : SINT := 1 ;					(* time offset in h for local time-zone (-12..+12) i.e. +1 for Berlin *)
	xSummerWinterTime : BOOL := TRUE  ;	(* consider Summertime from last sunday of march at 02:00 a.m.GMT to last sunday of october at 02:00 a.m.GMT *)
END_VAR

VAR_OUTPUT
	xActive : BOOL ;							(* server active, waiting for an request *)
	uiCountOfRequest : UINT ;				(* count of requests from a client *)
	sTimeClientIPAddress : STRING ;	(* IP address of the last client request *)
	xError : BOOL ;							(* last start or request generate an error - look "uiErrornumber" for reason *)
	uiErrorNumber : UINT ;					(* reason for the last error
		0 = No error
		1 = Ethernet socket could not opend 
		2 = Ethernet socket could not binded
		3 = Transmit time answer error
		4 = Ethernet receive error *)
END_VAR

VAR
	iSocketIndex : INT ;
	xBindSocket : BOOL ;

	diTraNr : DINT ;

	struSOCKADDRESS_Client : SOCKADDRESS ;
	diRecNr : DINT ;
	diIO : DINT ;
	dwParameterIO : DWORD ;
	arReceiveData : ARRAY[0..3] OF BYTE ;
	xSockInetNtoa : BOOL ;
	struInADDR_Client : INADDR;
	struSOCKADDRESS_Local : SOCKADDRESS ;
	uiLocalPort : UINT := 37 ;


	dtDateTime : DT ;
	uiSecond : UINT ;
	uiMinute : UINT ;
	uiHour : UINT ;
	uiDay : UINT ;
	uiMonth : UINT ;
	uiYear :UINT ;
	uiDayOfWeek : UINT ;
	xSummerTime : BOOL ;

	i : USINT ;

	Split_DT : NetTime_Split_DT ;

	uiDayStartSummertime : UINT ;
	uiDayEndSummertime : UINT ;
	dtStartSummertime : DT ;
	dtEndSummertime : DT ;

	udiGMTSecondsSince1900 : UDINT ;
	ptrSendData : POINTER TO ARRAY[0..3] OF BYTE ;
	arSendData : ARRAY[0..3] OF BYTE ;
	dwSendData : DWORD ;


END_VAR

IF xActive THEN
	IF xEnable THEN
		IF NetTime_ar_udiSockets[iSocketIndex] > 0 THEN
			(* waiting for an request.  Is any data received? *)
			diIO := SysSockIoctl(NetTime_ar_udiSockets[iSocketIndex], SOCKET_FIONREAD, ADR(dwParameterIO)); (* get num chars available to read *)
			IF dwParameterIO <> 0 THEN
				diRecNr := SysSockRecvFrom(NetTime_ar_udiSockets[iSocketIndex], ADR(arReceiveData), SIZEOF(arReceiveData), 0,
												 ADR(struSOCKADDRESS_Client), SIZEOF(struSOCKADDRESS_Client));
				IF diRecNr = -1 THEN
					uiErrorNumber := 4 ;
					xActive := FALSE ;
					NetTime_SockClose(iSocketIndex) ;
				ELSE
					uiCountOfRequest := uiCountOfRequest + 1 ;
					(* check receive IP Address *)
					struInADDR_Client.s_addr := struSOCKADDRESS_Client.sin_addr ;
					xSockInetNtoa:=SysSockInetNtoa(struInADDR_Client, sTimeClientIPAddress, SIZEOF(sTimeClientIPAddress)) ;

					(* get local real time clock *)
					dtDateTime :=SysRtcGetTime(TRUE) ;

					(* sub GMTOffset to get GMT *)
					dtDateTime := UDINT_TO_DT(DT_TO_UDINT(dtDateTime)-(DINT#3600*SINT_TO_DINT(siGMTOffset))) ;

					Split_DT(
						InputDT:=dtDateTime ,
						uiSecond=>uiSecond ,
						uiMinute=>uiMinute ,
						uiHour=>uiHour ,
						uiDay=>uiDay ,
						uiMonth=>uiMonth ,
						uiYear=>uiYear );

					uiDayOfWeek := NetTime_DayOfWeek(uiDay,uiMonth,uiYear) ;

					IF xSummerWinterTime THEN
						(* check if the actual time is in summertime interval
						last sunday of march at 2:00 a.m. to last sunday of october at 2:00 a.m. *)
						uiDayStartSummertime := 31-NetTime_DayOfWeek(31,3,uiYear) ;
						uiDayEndSummertime := 31-NetTime_DayOfWeek(31,10,uiYear) ;
						dtStartSummertime := NetTime_Concat_DT(0,0,2,uiDayStartSummertime,3,uiYear) ;
						dtEndSummertime := NetTime_Concat_DT(0,0,2,uiDayEndSummertime,10,uiYear) ;
						xSummerTime := (dtDateTime>dtStartSummertime) AND (dtDateTime<dtEndSummertime) ;
						IF xSummerTime THEN
							(* sub 1 hour to get GMT time *)
							dtDateTime := UDINT_TO_DT(DT_TO_UDINT(dtDateTime) - UDINT#3600) ;
							Split_DT(
								InputDT:=dtDateTime ,
								uiSecond=>uiSecond ,
								uiMinute=>uiMinute ,
								uiHour=>uiHour ,
								uiDay=>uiDay ,
								uiMonth=>uiMonth ,
								uiYear=>uiYear );
						END_IF
					END_IF

					udiGMTSecondsSince1900 := DT_TO_UDINT(dtDateTime) + UDINT#2208988800 ;

					ptrSendData := ADR(udiGMTSecondsSince1900) ;
					arSendData := ptrSendData^ ;

					(* change byte orientation *)
					dwSendData := 0 ;
					FOR i := 0 TO 3 DO
						dwSendData := SHL(dwSendData,8) ;
						dwSendData := dwSendData OR BYTE_TO_DWORD(arSendData[i]) ;
					END_FOR

					diTraNr := SysSockSendTo(NetTime_ar_udiSockets[iSocketIndex] , ADR(dwSendData), 4,0,
								ADR(struSOCKADDRESS_Client), SIZEOF(struSOCKADDRESS_Client));
					IF diTraNr < 0 THEN
						uiErrorNumber := 3 ;
						xActive := FALSE ;
						NetTime_SockClose(iSocketIndex) ;
					END_IF
				END_IF
			END_IF
		ELSE
			(* Socketindex is no longer valid! Perhaps PLC has stopt and socket has closed *)
			xActive := FALSE ;
			uiCountOfRequest := 0 ;
			sTimeClientIPAddress := '' ;
			xError := FALSE ;
			uiErrorNumber := 0 ;
		END_IF
	ELSE
		(* stop time server *)
		NetTime_SockClose(iSocketIndex) ;
		xActive := FALSE ;
		uiCountOfRequest := 0 ;
		sTimeClientIPAddress := '' ;
		xError := FALSE ;
		uiErrorNumber := 0 ;
	END_IF
ELSE
	IF xEnable THEN
		IF NOT xError THEN
			(* start timeserver *)
			xError := FALSE ;
			uiErrorNumber := 0;

			(* create a new  datagram-socket *)
			iSocketIndex := NetTime_SockCreate(SOCKET_AF_INET,SOCKET_DGRAM,0);
			IF iSocketIndex > 0 THEN
				(* Bind the socket to the local port *)
				struSOCKADDRESS_Local.sin_family := SOCKET_AF_INET; (* internetwork: UDP, TCP, etc. *)
				struSOCKADDRESS_Local.sin_addr := SysSockHtonl(SOCKET_INADDR_ANY) ;
				struSOCKADDRESS_Local.sin_port := SysSockHtons(uiLocalPort);
				xBindSocket := SysSockBind(NetTime_ar_udiSockets[iSocketIndex], ADR(struSOCKADDRESS_Local), SIZEOF(struSOCKADDRESS_Local));
				IF  NOT xBindSocket THEN
					NetTime_SockClose(iSocketIndex);
					uiErrorNumber := 2 ;
				ELSE
					xActive := TRUE ;
				END_IF
			ELSE
				uiErrorNumber := 1 ;
				NetTime_SockClose(iSocketIndex);
			END_IF
		END_IF
	ELSE
		(* reset last error *)
		uiCountOfRequest := 0 ;
		sTimeClientIPAddress := '' ;
		xError := FALSE ;
		uiErrorNumber := 0 ;
	END_IF
END_IF

xError := uiErrorNumber<>0 ;

END_FUNCTION_BLOCK

// XV300/Application/POUs/NetTime_RFC868_Server
FUNCTION_BLOCK NetTime_RFC868_Server (* prefix: srv868 *)
(* this FB is a server for time request from a client using a protocol described in RFC868 UDP *)
VAR_INPUT
	xEnable : BOOL ;							(* TRUE enable the server if there are no error, FALSE stop it and reset error *)
	siGMTOffset : SINT := 1 ;					(* time offset in h for local time-zone (-12..+12) i.e. +1 for Berlin *)
	xSummerWinterTime : BOOL := TRUE  ;	(* consider Summertime from last sunday of march at 02:00 a.m.GMT to last sunday of october at 02:00 a.m.GMT *)
END_VAR

VAR_OUTPUT
	xActive : BOOL ;							(* server active, waiting for an request *)
	uiCountOfRequest : UINT ;				(* count of requests from a client *)
	sTimeClientIPAddress : STRING ;	(* IP address of the last client request *)
	xError : BOOL ;							(* last start or request generate an error - look "uiErrornumber" for reason *)
	uiErrorNumber : UINT ;					(* reason for the last error
		0 = No error
		1 = Ethernet socket could not opend 
		2 = Ethernet socket could not binded
		3 = Transmit time answer error
		4 = Ethernet receive error *)
END_VAR

VAR
	iSocketIndex : INT ;
	xBindSocket : BOOL ;

	diTraNr : DINT ;

	struSOCKADDRESS_Client : SOCKADDRESS ;
	diRecNr : DINT ;
	diIO : DINT ;
	dwParameterIO : DWORD ;
	arReceiveData : ARRAY[0..3] OF BYTE ;
	xSockInetNtoa : BOOL ;
	struInADDR_Client : INADDR;
	struSOCKADDRESS_Local : SOCKADDRESS ;
	uiLocalPort : UINT := 37 ;


	dtDateTime : DT ;
	uiSecond : UINT ;
	uiMinute : UINT ;
	uiHour : UINT ;
	uiDay : UINT ;
	uiMonth : UINT ;
	uiYear :UINT ;
	uiDayOfWeek : UINT ;
	xSummerTime : BOOL ;

	i : USINT ;

	Split_DT : NetTime_Split_DT ;

	uiDayStartSummertime : UINT ;
	uiDayEndSummertime : UINT ;
	dtStartSummertime : DT ;
	dtEndSummertime : DT ;

	udiGMTSecondsSince1900 : UDINT ;
	ptrSendData : POINTER TO ARRAY[0..3] OF BYTE ;
	arSendData : ARRAY[0..3] OF BYTE ;
	dwSendData : DWORD ;


END_VAR

IF xActive THEN
	IF xEnable THEN
		IF NetTime_ar_udiSockets[iSocketIndex] > 0 THEN
			(* waiting for an request.  Is any data received? *)
			diIO := SysSockIoctl(NetTime_ar_udiSockets[iSocketIndex], SOCKET_FIONREAD, ADR(dwParameterIO)); (* get num chars available to read *)
			IF dwParameterIO <> 0 THEN
				diRecNr := SysSockRecvFrom(NetTime_ar_udiSockets[iSocketIndex], ADR(arReceiveData), SIZEOF(arReceiveData), 0,
												 ADR(struSOCKADDRESS_Client), SIZEOF(struSOCKADDRESS_Client));
				IF diRecNr = -1 THEN
					uiErrorNumber := 4 ;
					xActive := FALSE ;
					NetTime_SockClose(iSocketIndex) ;
				ELSE
					uiCountOfRequest := uiCountOfRequest + 1 ;
					(* check receive IP Address *)
					struInADDR_Client.s_addr := struSOCKADDRESS_Client.sin_addr ;
					xSockInetNtoa:=SysSockInetNtoa(struInADDR_Client, sTimeClientIPAddress, SIZEOF(sTimeClientIPAddress)) ;

					(* get local real time clock *)
					dtDateTime :=SysRtcGetTime(TRUE) ;

					(* sub GMTOffset to get GMT *)
					dtDateTime := UDINT_TO_DT(DT_TO_UDINT(dtDateTime)-(DINT#3600*SINT_TO_DINT(siGMTOffset))) ;

					Split_DT(
						InputDT:=dtDateTime ,
						uiSecond=>uiSecond ,
						uiMinute=>uiMinute ,
						uiHour=>uiHour ,
						uiDay=>uiDay ,
						uiMonth=>uiMonth ,
						uiYear=>uiYear );

					uiDayOfWeek := NetTime_DayOfWeek(uiDay,uiMonth,uiYear) ;

					IF xSummerWinterTime THEN
						(* check if the actual time is in summertime interval
						last sunday of march at 2:00 a.m. to last sunday of october at 2:00 a.m. *)
						uiDayStartSummertime := 31-NetTime_DayOfWeek(31,3,uiYear) ;
						uiDayEndSummertime := 31-NetTime_DayOfWeek(31,10,uiYear) ;
						dtStartSummertime := NetTime_Concat_DT(0,0,2,uiDayStartSummertime,3,uiYear) ;
						dtEndSummertime := NetTime_Concat_DT(0,0,2,uiDayEndSummertime,10,uiYear) ;
						xSummerTime := (dtDateTime>dtStartSummertime) AND (dtDateTime<dtEndSummertime) ;
						IF xSummerTime THEN
							(* sub 1 hour to get GMT time *)
							dtDateTime := UDINT_TO_DT(DT_TO_UDINT(dtDateTime) - UDINT#3600) ;
							Split_DT(
								InputDT:=dtDateTime ,
								uiSecond=>uiSecond ,
								uiMinute=>uiMinute ,
								uiHour=>uiHour ,
								uiDay=>uiDay ,
								uiMonth=>uiMonth ,
								uiYear=>uiYear );
						END_IF
					END_IF

					udiGMTSecondsSince1900 := DT_TO_UDINT(dtDateTime) + UDINT#2208988800 ;

					ptrSendData := ADR(udiGMTSecondsSince1900) ;
					arSendData := ptrSendData^ ;

					(* change byte orientation *)
					dwSendData := 0 ;
					FOR i := 0 TO 3 DO
						dwSendData := SHL(dwSendData,8) ;
						dwSendData := dwSendData OR BYTE_TO_DWORD(arSendData[i]) ;
					END_FOR

					diTraNr := SysSockSendTo(NetTime_ar_udiSockets[iSocketIndex] , ADR(dwSendData), 4,0,
								ADR(struSOCKADDRESS_Client), SIZEOF(struSOCKADDRESS_Client));
					IF diTraNr < 0 THEN
						uiErrorNumber := 3 ;
						xActive := FALSE ;
						NetTime_SockClose(iSocketIndex) ;
					END_IF
				END_IF
			END_IF
		ELSE
			(* Socketindex is no longer valid! Perhaps PLC has stopt and socket has closed *)
			xActive := FALSE ;
			uiCountOfRequest := 0 ;
			sTimeClientIPAddress := '' ;
			xError := FALSE ;
			uiErrorNumber := 0 ;
		END_IF
	ELSE
		(* stop time server *)
		NetTime_SockClose(iSocketIndex) ;
		xActive := FALSE ;
		uiCountOfRequest := 0 ;
		sTimeClientIPAddress := '' ;
		xError := FALSE ;
		uiErrorNumber := 0 ;
	END_IF
ELSE
	IF xEnable THEN
		IF NOT xError THEN
			(* start timeserver *)
			xError := FALSE ;
			uiErrorNumber := 0;

			(* create a new  datagram-socket *)
			iSocketIndex := NetTime_SockCreate(SOCKET_AF_INET,SOCKET_DGRAM,0);
			IF iSocketIndex > 0 THEN
				(* Bind the socket to the local port *)
				struSOCKADDRESS_Local.sin_family := SOCKET_AF_INET; (* internetwork: UDP, TCP, etc. *)
				struSOCKADDRESS_Local.sin_addr := SysSockHtonl(SOCKET_INADDR_ANY) ;
				struSOCKADDRESS_Local.sin_port := SysSockHtons(uiLocalPort);
				xBindSocket := SysSockBind(NetTime_ar_udiSockets[iSocketIndex], ADR(struSOCKADDRESS_Local), SIZEOF(struSOCKADDRESS_Local));
				IF  NOT xBindSocket THEN
					NetTime_SockClose(iSocketIndex);
					uiErrorNumber := 2 ;
				ELSE
					xActive := TRUE ;
				END_IF
			ELSE
				uiErrorNumber := 1 ;
				NetTime_SockClose(iSocketIndex);
			END_IF
		END_IF
	ELSE
		(* reset last error *)
		uiCountOfRequest := 0 ;
		sTimeClientIPAddress := '' ;
		xError := FALSE ;
		uiErrorNumber := 0 ;
	END_IF
END_IF

xError := uiErrorNumber<>0 ;

END_FUNCTION_BLOCK
